LIN {X 0,Y 531.686,Z 941.292,A -85,B 0,C 180,E1 4384.403,E2 4384.403} C_VEL
LIN {X 0,Y 531.304,Z 953.867,A -85,B 0,C 180,E1 4387.483,E2 4387.483} C_VEL
LIN {X 0,Y 531.16,Z 959.735,A -85,B 0,C 180,E1 4390.034,E2 4390.034} C_VEL
LIN {X 0,Y 530.961,Z 961.944,A -85,B 0,C 180,E1 4393.431,E2 4393.431} C_VEL
LIN {X 0,Y 531.167,Z 959.168,A -85,B 0,C 180,E1 4396.197,E2 4396.197} C_VEL
LIN {X 0,Y 531.42,Z 951.627,A -85,B 0,C 180,E1 4399.095,E2 4399.095} C_VEL
LIN {X 0,Y 531.761,Z 938.386,A -85,B 0,C 180,E1 4402.021,E2 4402.021} C_VEL
LIN {X 0,Y 532.428,Z 919.705,A -85,B 0,C 180,E1 4404.691,E2 4404.691} C_VEL
LIN {X 0,Y 533.219,Z 897.252,A -85,B 0,C 180,E1 4406.846,E2 4406.846} C_VEL
LIN {X 0,Y 533.797,Z 871.722,A -85,B 0,C 180,E1 4408.476,E2 4408.476} C_VEL
LIN {X 0,Y 530.532,Z 857.28,A -85,B 0,C 180,E1 4409.284,E2 4409.284} C_VEL
LIN {X 0,Y 530.829,Z 857.28,A -85,B 0,C 180,E1 4414.908,E2 4414.908} C_VEL
LIN {X 0,Y 530.721,Z 857.28,A -85,B 0,C 180,E1 4419.855,E2 4419.855} C_VEL
LIN {X 0,Y 530.626,Z 857.28,A -85,B 0,C 180,E1 4424.88,E2 4424.88} C_VEL
LIN {X 0,Y 530.545,Z 857.28,A -85,B 0,C 180,E1 4430.026,E2 4430.026} C_VEL
LIN {X 0,Y 530.38,Z 857.28,A -85,B 0,C 180,E1 4435.353,E2 4435.353} C_VEL
LIN {X 0,Y 530.253,Z 857.28,A -85,B 0,C 180,E1 4441.143,E2 4441.143} C_VEL
LIN {X 0,Y 530.208,Z 857.28,A -85,B 0,C 180,E1 4446.978,E2 4446.978} C_VEL
LIN {X 0,Y 530.229,Z 857.28,A -85,B 0,C 180,E1 4453.26,E2 4453.26} C_VEL
LIN {X 0,Y 530.267,Z 857.28,A -85,B 0,C 180,E1 4458.999,E2 4458.999} C_VEL
LIN {X 0,Y 530.449,Z 857.934,A -85,B 0,C 180,E1 4461.861,E2 4461.861} C_VEL
LIN {X 0,Y 533.507,Z 877.785,A -85,B 0,C 180,E1 4462.888,E2 4462.888} C_VEL
LIN {X 0,Y 532.84,Z 903.715,A -85,B 0,C 180,E1 4464.706,E2 4464.706} C_VEL
LIN {X 0,Y 532.072,Z 925.667,A -85,B 0,C 180,E1 4467.04,E2 4467.04} C_VEL
LIN {X 0,Y 531.58,Z 942.941,A -85,B 0,C 180,E1 4469.823,E2 4469.823} C_VEL
LIN {X 0,Y 531.314,Z 954.833,A -85,B 0,C 180,E1 4472.91,E2 4472.91} C_VEL
LIN {X 0,Y 531.021,Z 960.608,A -85,B 0,C 180,E1 4475.838,E2 4475.838} C_VEL
LIN {X 0,Y 530.948,Z 961.777,A -85,B 0,C 180,E1 4478.273,E2 4478.273} C_VEL
LIN {X 0,Y 531.171,Z 959.373,A -85,B 0,C 180,E1 4480.97,E2 4480.97} C_VEL
LIN {X 0,Y 531.35,Z 952.112,A -85,B 0,C 180,E1 4483.898,E2 4483.898} C_VEL
LIN {X 0,Y 531.721,Z 939.03,A -85,B 0,C 180,E1 4486.86,E2 4486.86} C_VEL
LIN {X 0,Y 532.237,Z 921.058,A -85,B 0,C 180,E1 4489.473,E2 4489.473} C_VEL
LIN {X 0,Y 532.958,Z 898.658,A -85,B 0,C 180,E1 4491.653,E2 4491.653} C_VEL
LIN {X 0,Y 533.718,Z 872.183,A -85,B 0,C 180,E1 4493.332,E2 4493.332} C_VEL
LIN {X 0,Y 530.984,Z 857.28,A -85,B 0,C 180,E1 4494.148,E2 4494.148} C_VEL
LIN {X 0,Y 530.827,Z 857.28,A -85,B 0,C 180,E1 4500.021,E2 4500.021} C_VEL
LIN {X 0,Y 530.801,Z 857.28,A -85,B 0,C 180,E1 4504.928,E2 4504.928} C_VEL
LIN {X 0,Y 530.696,Z 857.28,A -85,B 0,C 180,E1 4509.873,E2 4509.873} C_VEL
LIN {X 0,Y 530.612,Z 857.28,A -85,B 0,C 180,E1 4514.896,E2 4514.896} C_VEL
LIN {X 0,Y 530.576,Z 857.28,A -85,B 0,C 180,E1 4520.039,E2 4520.039} C_VEL
LIN {X 0,Y 530.461,Z 857.28,A -85,B 0,C 180,E1 4525.361,E2 4525.361} C_VEL
LIN {X 0,Y 530.352,Z 857.28,A -85,B 0,C 180,E1 4527.012,E2 4527.012} C_VEL
LIN {X 0,Y 527.829,Z 857.28,A -85,B 0,C 180,E1 4528.404,E2 4528.404} C_VEL
LIN {X 0,Y 522.406,Z 857.28,A -85,B 0,C 180,E1 4530.49,E2 4530.49} C_VEL
LIN {X 0,Y 522.316,Z 857.28,A -85,B 0,C 180,E1 4530.731,E2 4530.731} C_VEL
LIN {X 0,Y 522.326,Z 857.28,A -85,B 0,C 180,E1 4535.744,E2 4535.744} C_VEL
LIN {X 0,Y 522.316,Z 857.28,A -85,B 0,C 180,E1 4541.821,E2 4541.821} C_VEL
LIN {X 0,Y 522.421,Z 857.28,A -85,B 0,C 180,E1 4548.197,E2 4548.197} C_VEL
LIN {X 0,Y 522.325,Z 857.28,A -85,B 0,C 180,E1 4554.568,E2 4554.568} C_VEL
LIN {X 0,Y 522.426,Z 857.28,A -85,B 0,C 180,E1 4560.483,E2 4560.483} C_VEL
LIN {X 0,Y 522.61,Z 857.28,A -85,B 0,C 180,E1 4564.312,E2 4564.312} C_VEL
LIN {X 0,Y 530.423,Z 879.508,A -85,B 0,C 180,E1 4565.071,E2 4565.071} C_VEL
LIN {X 0,Y 530.037,Z 939.927,A -85,B 0,C 180,E1 4566.073,E2 4566.073} C_VEL
LIN {X 0,Y 528.959,Z 972.429,A -85,B 0,C 180,E1 4567.213,E2 4567.213} C_VEL
LIN {X 0,Y 527.599,Z 1004.287,A -85,B 0,C 180,E1 4568.993,E2 4568.993} C_VEL
LIN {X 0,Y 526.123,Z 1033.257,A -85,B 0,C 180,E1 4571.328,E2 4571.328} C_VEL
LIN {X 0,Y 524.904,Z 1058.08,A -85,B 0,C 180,E1 4574.097,E2 4574.097} C_VEL
LIN {X 0,Y 523.978,Z 1078.839,A -85,B 0,C 180,E1 4577.272,E2 4577.272} C_VEL
LIN {X 0,Y 523.47,Z 1095.118,A -85,B 0,C 180,E1 4580.847,E2 4580.847} C_VEL
LIN {X 0,Y 523.252,Z 1104.993,A -85,B 0,C 180,E1 4584.188,E2 4584.188} C_VEL
LIN {X 0,Y 523.184,Z 1109.404,A -85,B 0,C 180,E1 4586.682,E2 4586.682} C_VEL
LIN {X 0,Y 523.198,Z 1111.5,A -85,B 0,C 180,E1 4590.001,E2 4590.001} C_VEL
LIN {X 0,Y 523.22,Z 1108.484,A -85,B 0,C 180,E1 4593.955,E2 4593.955} C_VEL
LIN {X 0,Y 523.378,Z 1100.701,A -85,B 0,C 180,E1 4597.481,E2 4597.481} C_VEL
LIN {X 0,Y 523.696,Z 1087.408,A -85,B 0,C 180,E1 4601.022,E2 4601.022} C_VEL
LIN {X 0,Y 524.459,Z 1068.424,A -85,B 0,C 180,E1 4604.456,E2 4604.456} C_VEL
LIN {X 0,Y 525.575,Z 1043.869,A -85,B 0,C 180,E1 4607.594,E2 4607.594} C_VEL
LIN {X 0,Y 526.962,Z 1015.854,A -85,B 0,C 180,E1 4610.169,E2 4610.169} C_VEL
LIN {X 0,Y 528.484,Z 984.528,A -85,B 0,C 180,E1 4612.199,E2 4612.199} C_VEL
LIN {X 0,Y 529.692,Z 950.575,A -85,B 0,C 180,E1 4613.623,E2 4613.623} C_VEL
LIN {X 0,Y 530.348,Z 915.537,A -85,B 0,C 180,E1 4614.406,E2 4614.406} C_VEL
LIN {X 0,Y 529.868,Z 878.299,A -85,B 0,C 180,E1 4614.974,E2 4614.974} C_VEL
LIN {X 0,Y 522.471,Z 857.28,A -85,B 0,C 180,E1 4615.766,E2 4615.766} C_VEL
LIN {X 0,Y 522.371,Z 857.28,A -85,B 0,C 180,E1 4621.449,E2 4621.449} C_VEL
LIN {X 0,Y 522.284,Z 857.28,A -85,B 0,C 180,E1 4627.502,E2 4627.502} C_VEL
LIN {X 0,Y 522.319,Z 857.28,A -85,B 0,C 180,E1 4633.552,E2 4633.552} C_VEL
LIN {X 0,Y 522.389,Z 857.28,A -85,B 0,C 180,E1 4638.902,E2 4638.902} C_VEL
LIN {X 0,Y 522.342,Z 857.28,A -85,B 0,C 180,E1 4644.56,E2 4644.56} C_VEL
LIN {X 0,Y 522.409,Z 857.28,A -85,B 0,C 180,E1 4650.471,E2 4650.471} C_VEL
LIN {X 0,Y 522.582,Z 857.28,A -85,B 0,C 180,E1 4656.058,E2 4656.058} C_VEL
LIN {X 0,Y 522.722,Z 857.28,A -85,B 0,C 180,E1 4661.407,E2 4661.407} C_VEL
LIN {X 0,Y 522.636,Z 857.28,A -85,B 0,C 180,E1 4668.283,E2 4668.283} C_VEL
LIN {X 0,Y 522.958,Z 857.28,A -85,B 0,C 180,E1 4673.331,E2 4673.331} C_VEL
LIN {X 0,Y 522.942,Z 857.28,A -85,B 0,C 180,E1 4679.979,E2 4679.979} C_VEL
LIN {X 0,Y 522.877,Z 857.28,A -85,B 0,C 180,E1 4684.96,E2 4684.96} C_VEL
LIN {X 0,Y 522.769,Z 857.28,A -85,B 0,C 180,E1 4690.022,E2 4690.022} C_VEL
LIN {X 0,Y 522.692,Z 857.28,A -85,B 0,C 180,E1 4695.083,E2 4695.083} C_VEL
LIN {X 0,Y 522.637,Z 857.28,A -85,B 0,C 180,E1 4700.311,E2 4700.311} C_VEL
LIN {X 0,Y 522.478,Z 857.28,A -85,B 0,C 180,E1 4706.058,E2 4706.058} C_VEL
LIN {X 0,Y 522.342,Z 857.28,A -85,B 0,C 180,E1 4711.41,E2 4711.41} C_VEL
LIN {X 0,Y 522.255,Z 857.28,A -85,B 0,C 180,E1 4717.458,E2 4717.458} C_VEL
LIN {X 0,Y 522.35,Z 857.28,A -85,B 0,C 180,E1 4723.56,E2 4723.56} C_VEL
LIN {X 0,Y 522.376,Z 857.28,A -85,B 0,C 180,E1 4728.842,E2 4728.842} C_VEL
LIN {X 0,Y 522.429,Z 857.28,A -85,B 0,C 180,E1 4734.575,E2 4734.575} C_VEL
LIN {X 0,Y 522.636,Z 857.79,A -85,B 0,C 180,E1 4736.295,E2 4736.295} C_VEL
LIN {X 0,Y 526.502,Z 877.686,A -85,B 0,C 180,E1 4737.414,E2 4737.414} C_VEL
LIN {X 0,Y 525.643,Z 903.07,A -85,B 0,C 180,E1 4739.199,E2 4739.199} C_VEL
LIN {X 0,Y 524.669,Z 924.663,A -85,B 0,C 180,E1 4741.464,E2 4741.464} C_VEL
LIN {X 0,Y 524.04,Z 941.697,A -85,B 0,C 180,E1 4744.104,E2 4744.104} C_VEL
LIN {X 0,Y 523.64,Z 953.648,A -85,B 0,C 180,E1 4746.937,E2 4746.937} C_VEL
LIN {X 0,Y 523.4,Z 960.427,A -85,B 0,C 180,E1 4749.687,E2 4749.687} C_VEL
LIN {X 0,Y 523.152,Z 963.153,A -85,B 0,C 180,E1 4752.608,E2 4752.608} C_VEL
LIN {X 0,Y 523.311,Z 961.505,A -85,B 0,C 180,E1 4755.481,E2 4755.481} C_VEL
LIN {X 0,Y 523.516,Z 955.588,A -85,B 0,C 180,E1 4758.319,E2 4758.319} C_VEL
LIN {X 0,Y 523.978,Z 943.155,A -85,B 0,C 180,E1 4761.483,E2 4761.483} C_VEL
LIN {X 0,Y 524.612,Z 925.67,A -85,B 0,C 180,E1 4764.282,E2 4764.282} C_VEL
LIN {X 0,Y 525.495,Z 904.106,A -85,B 0,C 180,E1 4766.593,E2 4766.593} C_VEL
LIN {X 0,Y 526.42,Z 879.629,A -85,B 0,C 180,E1 4768.351,E2 4768.351} C_VEL
LIN {X 0,Y 524.585,Z 865.354,A -85,B 0,C 180,E1 4769.173,E2 4769.173} C_VEL
LIN {X 0,Y 522.578,Z 857.28,A -85,B 0,C 180,E1 4769.688,E2 4769.688} C_VEL
LIN {X 0,Y 522.915,Z 857.28,A -85,B 0,C 180,E1 4774.983,E2 4774.983} C_VEL
LIN {X 0,Y 522.774,Z 857.28,A -85,B 0,C 180,E1 4780.288,E2 4780.288} C_VEL
LIN {X 0,Y 522.689,Z 857.28,A -85,B 0,C 180,E1 4785.111,E2 4785.111} C_VEL
LIN {X 0,Y 522.592,Z 857.28,A -85,B 0,C 180,E1 4790.344,E2 4790.344} C_VEL
LIN {X 0,Y 522.426,Z 857.28,A -85,B 0,C 180,E1 4796.146,E2 4796.146} C_VEL
LIN {X 0,Y 522.344,Z 857.28,A -85,B 0,C 180,E1 4801.449,E2 4801.449} C_VEL
LIN {X 0,Y 522.245,Z 857.28,A -85,B 0,C 180,E1 4807.504,E2 4807.504} C_VEL
LIN {X 0,Y 522.328,Z 857.28,A -85,B 0,C 180,E1 4813.615,E2 4813.615} C_VEL
LIN {X 0,Y 522.374,Z 857.28,A -85,B 0,C 180,E1 4818.902,E2 4818.902} C_VEL
LIN {X 0,Y 522.476,Z 857.505,A -85,B 0,C 180,E1 4821.573,E2 4821.573} C_VEL
LIN {X 0,Y 525.93,Z 878.07,A -85,B 0,C 180,E1 4822.641,E2 4822.641} C_VEL
LIN {X 0,Y 525.266,Z 903.689,A -85,B 0,C 180,E1 4824.434,E2 4824.434} C_VEL
LIN {X 0,Y 524.418,Z 925.824,A -85,B 0,C 180,E1 4826.773,E2 4826.773} C_VEL
LIN {X 0,Y 523.86,Z 942.873,A -85,B 0,C 180,E1 4829.473,E2 4829.473} C_VEL
LIN {X 0,Y 523.539,Z 954.889,A -85,B 0,C 180,E1 4832.474,E2 4832.474} C_VEL
LIN {X 0,Y 523.261,Z 961.323,A -85,B 0,C 180,E1 4835.456,E2 4835.456} C_VEL
LIN {X 0,Y 523.151,Z 963.019,A -85,B 0,C 180,E1 4837.932,E2 4837.932} C_VEL
LIN {X 0,Y 523.343,Z 961.014,A -85,B 0,C 180,E1 4840.722,E2 4840.722} C_VEL
LIN {X 0,Y 523.558,Z 954.393,A -85,B 0,C 180,E1 4843.652,E2 4843.652} C_VEL
LIN {X 0,Y 523.892,Z 942.002,A -85,B 0,C 180,E1 4846.66,E2 4846.66} C_VEL
LIN {X 0,Y 524.514,Z 924.374,A -85,B 0,C 180,E1 4849.37,E2 4849.37} C_VEL
LIN {X 0,Y 525.279,Z 902.377,A -85,B 0,C 180,E1 4851.634,E2 4851.634} C_VEL
LIN {X 0,Y 526.144,Z 877.428,A -85,B 0,C 180,E1 4853.325,E2 4853.325} C_VEL
LIN {X 0,Y 523.03,Z 857.28,A -85,B 0,C 180,E1 4854.417,E2 4854.417} C_VEL
LIN {X 0,Y 522.945,Z 857.28,A -85,B 0,C 180,E1 4860.021,E2 4860.021} C_VEL
LIN {X 0,Y 522.887,Z 857.28,A -85,B 0,C 180,E1 4865.003,E2 4865.003} C_VEL
LIN {X 0,Y 522.792,Z 857.28,A -85,B 0,C 180,E1 4870.043,E2 4870.043} C_VEL
LIN {X 0,Y 522.676,Z 857.28,A -85,B 0,C 180,E1 4875.127,E2 4875.127} C_VEL
LIN {X 0,Y 522.636,Z 857.28,A -85,B 0,C 180,E1 4880.356,E2 4880.356} C_VEL
LIN {X 0,Y 522.462,Z 857.28,A -85,B 0,C 180,E1 4886.057,E2 4886.057} C_VEL
LIN {X 0,Y 522.316,Z 857.28,A -85,B 0,C 180,E1 4890.731,E2 4890.731} C_VEL
LIN {X 0,Y 519.814,Z 857.28,A -85,B 0,C 180,E1 4892.139,E2 4892.139} C_VEL
LIN {X 0,Y 514.508,Z 857.28,A -85,B 0,C 180,E1 4894.249,E2 4894.249} C_VEL
LIN {X 0,Y 514.42,Z 857.28,A -85,B 0,C 180,E1 4894.493,E2 4894.493} C_VEL
LIN {X 0,Y 514.38,Z 857.28,A -85,B 0,C 180,E1 4900.366,E2 4900.366} C_VEL
LIN {X 0,Y 514.435,Z 857.28,A -85,B 0,C 180,E1 4905.061,E2 4905.061} C_VEL
LIN {X 0,Y 514.493,Z 857.28,A -85,B 0,C 180,E1 4909.924,E2 4909.924} C_VEL
LIN {X 0,Y 514.394,Z 857.28,A -85,B 0,C 180,E1 4915.997,E2 4915.997} C_VEL
LIN {X 0,Y 514.572,Z 857.28,A -85,B 0,C 180,E1 4921.972,E2 4921.972} C_VEL
LIN {X 0,Y 514.678,Z 857.28,A -85,B 0,C 180,E1 4923.935,E2 4923.935} C_VEL
LIN {X 0,Y 523.207,Z 881.258,A -85,B 0,C 180,E1 4924.73,E2 4924.73} C_VEL
LIN {X 0,Y 522.815,Z 939.926,A -85,B 0,C 180,E1 4925.722,E2 4925.722} C_VEL
LIN {X 0,Y 521.638,Z 972.428,A -85,B 0,C 180,E1 4926.875,E2 4926.875} C_VEL
LIN {X 0,Y 520.147,Z 1004.749,A -85,B 0,C 180,E1 4928.711,E2 4928.711} C_VEL
LIN {X 0,Y 518.481,Z 1034.401,A -85,B 0,C 180,E1 4931.153,E2 4931.153} C_VEL
LIN {X 0,Y 517.127,Z 1059.679,A -85,B 0,C 180,E1 4934.069,E2 4934.069} C_VEL
LIN {X 0,Y 516.104,Z 1081.097,A -85,B 0,C 180,E1 4937.505,E2 4937.505} C_VEL
LIN {X 0,Y 515.593,Z 1096.65,A -85,B 0,C 180,E1 4941.132,E2 4941.132} C_VEL
LIN {X 0,Y 515.398,Z 1106.726,A -85,B 0,C 180,E1 4944.945,E2 4944.945} C_VEL
LIN {X 0,Y 515.284,Z 1110.932,A -85,B 0,C 180,E1 4948.317,E2 4948.317} C_VEL
LIN {X 0,Y 515.293,Z 1110.931,A -85,B 0,C 180,E1 4951.684,E2 4951.684} C_VEL
LIN {X 0,Y 515.399,Z 1106.723,A -85,B 0,C 180,E1 4955.057,E2 4955.057} C_VEL
LIN {X 0,Y 515.605,Z 1096.648,A -85,B 0,C 180,E1 4958.869,E2 4958.869} C_VEL
LIN {X 0,Y 516.101,Z 1081.092,A -85,B 0,C 180,E1 4962.496,E2 4962.496} C_VEL
LIN {X 0,Y 517.137,Z 1059.67,A -85,B 0,C 180,E1 4965.932,E2 4965.932} C_VEL
LIN {X 0,Y 518.503,Z 1034.387,A -85,B 0,C 180,E1 4968.847,E2 4968.847} C_VEL
LIN {X 0,Y 520.158,Z 1004.698,A -85,B 0,C 180,E1 4971.292,E2 4971.292} C_VEL
LIN {X 0,Y 521.592,Z 972.395,A -85,B 0,C 180,E1 4973.129,E2 4973.129} C_VEL
LIN {X 0,Y 522.793,Z 937.798,A -85,B 0,C 180,E1 4974.341,E2 4974.341} C_VEL
LIN {X 0,Y 522.824,Z 880.394,A -85,B 0,C 180,E1 4975.303,E2 4975.303} C_VEL
LIN {X 0,Y 514.56,Z 857.28,A -85,B 0,C 180,E1 4976.12,E2 4976.12} C_VEL
LIN {X 0,Y 514.453,Z 857.28,A -85,B 0,C 180,E1 4981.99,E2 4981.99} C_VEL
LIN {X 0,Y 514.363,Z 857.28,A -85,B 0,C 180,E1 4988.182,E2 4988.182} C_VEL
LIN {X 0,Y 514.366,Z 857.28,A -85,B 0,C 180,E1 4992.612,E2 4992.612} C_VEL
LIN {X 0,Y 514.446,Z 857.28,A -85,B 0,C 180,E1 4997.39,E2 4997.39} C_VEL
LIN {X 0,Y 514.434,Z 857.28,A -85,B 0,C 180,E1 5002.624,E2 5002.624} C_VEL
LIN {X 0,Y 514.48,Z 857.28,A -85,B 0,C 180,E1 5008.59,E2 5008.59} C_VEL
LIN {X 0,Y 514.578,Z 857.28,A -85,B 0,C 180,E1 5013.798,E2 5013.798} C_VEL
LIN {X 0,Y 514.739,Z 857.28,A -85,B 0,C 180,E1 5020.267,E2 5020.267} C_VEL
LIN {X 0,Y 514.565,Z 857.28,A -85,B 0,C 180,E1 5026.172,E2 5026.172} C_VEL
LIN {X 0,Y 514.82,Z 857.28,A -85,B 0,C 180,E1 5031.526,E2 5031.526} C_VEL
LIN {X 0,Y 514.981,Z 857.28,A -85,B 0,C 180,E1 5036.609,E2 5036.609} C_VEL
LIN {X 0,Y 514.972,Z 857.28,A -85,B 0,C 180,E1 5041.663,E2 5041.663} C_VEL
LIN {X 0,Y 514.904,Z 857.28,A -85,B 0,C 180,E1 5046.73,E2 5046.73} C_VEL
LIN {X 0,Y 514.781,Z 857.28,A -85,B 0,C 180,E1 5051.854,E2 5051.854} C_VEL
LIN {X 0,Y 514.737,Z 857.28,A -85,B 0,C 180,E1 5057.076,E2 5057.076} C_VEL
LIN {X 0,Y 514.634,Z 857.28,A -85,B 0,C 180,E1 5062.453,E2 5062.453} C_VEL
LIN {X 0,Y 514.526,Z 857.28,A -85,B 0,C 180,E1 5068.05,E2 5068.05} C_VEL
LIN {X 0,Y 514.385,Z 857.28,A -85,B 0,C 180,E1 5073.962,E2 5073.962} C_VEL
LIN {X 0,Y 514.382,Z 857.28,A -85,B 0,C 180,E1 5080.309,E2 5080.309} C_VEL
LIN {X 0,Y 514.406,Z 857.28,A -85,B 0,C 180,E1 5085.056,E2 5085.056} C_VEL
LIN {X 0,Y 514.464,Z 857.28,A -85,B 0,C 180,E1 5091.827,E2 5091.827} C_VEL
LIN {X 0,Y 514.722,Z 857.28,A -85,B 0,C 180,E1 5095.905,E2 5095.905} C_VEL
LIN {X 0,Y 519.052,Z 878.103,A -85,B 0,C 180,E1 5097.103,E2 5097.103} C_VEL
LIN {X 0,Y 518.142,Z 903.526,A -85,B 0,C 180,E1 5098.901,E2 5098.901} C_VEL
LIN {X 0,Y 517.103,Z 925.104,A -85,B 0,C 180,E1 5101.175,E2 5101.175} C_VEL
LIN {X 0,Y 516.343,Z 942.645,A -85,B 0,C 180,E1 5103.905,E2 5103.905} C_VEL
LIN {X 0,Y 515.932,Z 954.252,A -85,B 0,C 180,E1 5106.66,E2 5106.66} C_VEL
LIN {X 0,Y 515.589,Z 962.018,A -85,B 0,C 180,E1 5109.872,E2 5109.872} C_VEL
LIN {X 0,Y 515.372,Z 964.38,A -85,B 0,C 180,E1 5112.915,E2 5112.915} C_VEL
LIN {X 0,Y 515.584,Z 961.302,A -85,B 0,C 180,E1 5116.412,E2 5116.412} C_VEL
LIN {X 0,Y 515.929,Z 953.427,A -85,B 0,C 180,E1 5119.443,E2 5119.443} C_VEL
LIN {X 0,Y 516.389,Z 940.148,A -85,B 0,C 180,E1 5122.418,E2 5122.418} C_VEL
LIN {X 0,Y 517.248,Z 921.213,A -85,B 0,C 180,E1 5125.172,E2 5125.172} C_VEL
LIN {X 0,Y 518.229,Z 898.544,A -85,B 0,C 180,E1 5127.383,E2 5127.383} C_VEL
LIN {X 0,Y 518.522,Z 873.107,A -85,B 0,C 180,E1 5129.058,E2 5129.058} C_VEL
LIN {X 0,Y 514.633,Z 857.28,A -85,B 0,C 180,E1 5129.999,E2 5129.999} C_VEL
LIN {X 0,Y 515.018,Z 857.28,A -85,B 0,C 180,E1 5135.059,E2 5135.059} C_VEL
LIN {X 0,Y 514.896,Z 857.28,A -85,B 0,C 180,E1 5140.161,E2 5140.161} C_VEL
LIN {X 0,Y 514.751,Z 857.28,A -85,B 0,C 180,E1 5145.35,E2 5145.35} C_VEL
LIN {X 0,Y 514.648,Z 857.28,A -85,B 0,C 180,E1 5150.673,E2 5150.673} C_VEL
LIN {X 0,Y 514.546,Z 857.28,A -85,B 0,C 180,E1 5156.191,E2 5156.191} C_VEL
LIN {X 0,Y 514.428,Z 857.28,A -85,B 0,C 180,E1 5161.99,E2 5161.99} C_VEL
LIN {X 0,Y 514.344,Z 857.28,A -85,B 0,C 180,E1 5168.183,E2 5168.183} C_VEL
LIN {X 0,Y 514.394,Z 857.28,A -85,B 0,C 180,E1 5174.944,E2 5174.944} C_VEL
LIN {X 0,Y 514.622,Z 858.024,A -85,B 0,C 180,E1 5181.318,E2 5181.318} C_VEL
LIN {X 0,Y 518.349,Z 879.334,A -85,B 0,C 180,E1 5182.443,E2 5182.443} C_VEL
LIN {X 0,Y 517.635,Z 904.658,A -85,B 0,C 180,E1 5184.242,E2 5184.242} C_VEL
LIN {X 0,Y 516.804,Z 925.31,A -85,B 0,C 180,E1 5186.416,E2 5186.416} C_VEL
LIN {X 0,Y 516.172,Z 941.896,A -85,B 0,C 180,E1 5188.955,E2 5188.955} C_VEL
LIN {X 0,Y 515.766,Z 954.888,A -85,B 0,C 180,E1 5192.023,E2 5192.023} C_VEL
LIN {X 0,Y 515.548,Z 961.578,A -85,B 0,C 180,E1 5194.804,E2 5194.804} C_VEL
LIN {X 0,Y 515.323,Z 964.146,A -85,B 0,C 180,E1 5197.579,E2 5197.579} C_VEL
LIN {X 0,Y 515.481,Z 963.124,A -85,B 0,C 180,E1 5200.034,E2 5200.034} C_VEL
LIN {X 0,Y 515.741,Z 957.805,A -85,B 0,C 180,E1 5202.958,E2 5202.958} C_VEL
LIN {X 0,Y 516.086,Z 947.027,A -85,B 0,C 180,E1 5206,E2 5206} C_VEL
LIN {X 0,Y 516.68,Z 930.919,A -85,B 0,C 180,E1 5208.812,E2 5208.812} C_VEL
LIN {X 0,Y 517.521,Z 909.442,A -85,B 0,C 180,E1 5211.296,E2 5211.296} C_VEL
LIN {X 0,Y 518.354,Z 885.382,A -85,B 0,C 180,E1 5213.144,E2 5213.144} C_VEL
LIN {X 0,Y 517.545,Z 868.672,A -85,B 0,C 180,E1 5214.076,E2 5214.076} C_VEL
LIN {X 0,Y 515.108,Z 857.28,A -85,B 0,C 180,E1 5214.656,E2 5214.656} C_VEL
LIN {X 0,Y 515.044,Z 857.28,A -85,B 0,C 180,E1 5220.022,E2 5220.022} C_VEL
LIN {X 0,Y 514.98,Z 857.28,A -85,B 0,C 180,E1 5225.08,E2 5225.08} C_VEL
LIN {X 0,Y 514.896,Z 857.28,A -85,B 0,C 180,E1 5230.179,E2 5230.179} C_VEL
LIN {X 0,Y 514.767,Z 857.28,A -85,B 0,C 180,E1 5235.366,E2 5235.366} C_VEL
LIN {X 0,Y 514.701,Z 857.28,A -85,B 0,C 180,E1 5240.685,E2 5240.685} C_VEL
LIN {X 0,Y 514.557,Z 857.28,A -85,B 0,C 180,E1 5246.203,E2 5246.203} C_VEL
LIN {X 0,Y 514.462,Z 857.28,A -85,B 0,C 180,E1 5251.998,E2 5251.998} C_VEL
LIN {X 0,Y 514.42,Z 857.28,A -85,B 0,C 180,E1 5254.493,E2 5254.493} C_VEL
LIN {X 0,Y 511.854,Z 857.28,A -85,B 0,C 180,E1 5255.93,E2 5255.93} C_VEL
LIN {X 0,Y 506.441,Z 857.28,A -85,B 0,C 180,E1 5258.083,E2 5258.083} C_VEL
LIN {X 0,Y 506.357,Z 857.28,A -85,B 0,C 180,E1 5258.333,E2 5258.333} C_VEL
LIN {X 0,Y 506.432,Z 857.28,A -85,B 0,C 180,E1 5264.15,E2 5264.15} C_VEL
LIN {X 0,Y 506.496,Z 857.28,A -85,B 0,C 180,E1 5268.88,E2 5268.88} C_VEL
LIN {X 0,Y 506.484,Z 857.28,A -85,B 0,C 180,E1 5275.391,E2 5275.391} C_VEL
LIN {X 0,Y 506.589,Z 857.28,A -85,B 0,C 180,E1 5281.433,E2 5281.433} C_VEL
LIN {X 0,Y 506.719,Z 857.28,A -85,B 0,C 180,E1 5283.563,E2 5283.563} C_VEL
LIN {X 0,Y 516.179,Z 885.355,A -85,B 0,C 180,E1 5284.423,E2 5284.423} C_VEL
LIN {X 0,Y 515.581,Z 941.148,A -85,B 0,C 180,E1 5285.394,E2 5285.394} C_VEL
LIN {X 0,Y 514.28,Z 974.856,A -85,B 0,C 180,E1 5286.639,E2 5286.639} C_VEL
LIN {X 0,Y 512.594,Z 1006.805,A -85,B 0,C 180,E1 5288.534,E2 5288.534} C_VEL
LIN {X 0,Y 510.831,Z 1035.498,A -85,B 0,C 180,E1 5290.972,E2 5290.972} C_VEL
LIN {X 0,Y 509.354,Z 1061.277,A -85,B 0,C 180,E1 5294.041,E2 5294.041} C_VEL
LIN {X 0,Y 508.243,Z 1082.183,A -85,B 0,C 180,E1 5297.528,E2 5297.528} C_VEL
LIN {X 0,Y 507.722,Z 1096.65,A -85,B 0,C 180,E1 5300.993,E2 5300.993} C_VEL
LIN {X 0,Y 507.492,Z 1106.725,A -85,B 0,C 180,E1 5304.866,E2 5304.866} C_VEL
LIN {X 0,Y 507.401,Z 1110.932,A -85,B 0,C 180,E1 5308.291,E2 5308.291} C_VEL
LIN {X 0,Y 507.409,Z 1110.931,A -85,B 0,C 180,E1 5311.711,E2 5311.711} C_VEL
LIN {X 0,Y 507.493,Z 1106.723,A -85,B 0,C 180,E1 5315.136,E2 5315.136} C_VEL
LIN {X 0,Y 507.735,Z 1096.648,A -85,B 0,C 180,E1 5319.008,E2 5319.008} C_VEL
LIN {X 0,Y 508.286,Z 1081.092,A -85,B 0,C 180,E1 5322.691,E2 5322.691} C_VEL
LIN {X 0,Y 509.414,Z 1059.67,A -85,B 0,C 180,E1 5326.18,E2 5326.18} C_VEL
LIN {X 0,Y 510.931,Z 1034.388,A -85,B 0,C 180,E1 5329.137,E2 5329.137} C_VEL
LIN {X 0,Y 512.698,Z 1005.302,A -85,B 0,C 180,E1 5331.573,E2 5331.573} C_VEL
LIN {X 0,Y 514.308,Z 972.393,A -85,B 0,C 180,E1 5333.476,E2 5333.476} C_VEL
LIN {X 0,Y 515.627,Z 937.222,A -85,B 0,C 180,E1 5334.717,E2 5334.717} C_VEL
LIN {X 0,Y 515.82,Z 882.841,A -85,B 0,C 180,E1 5335.633,E2 5335.633} C_VEL
LIN {X 0,Y 506.612,Z 857.28,A -85,B 0,C 180,E1 5336.511,E2 5336.511} C_VEL
LIN {X 0,Y 506.479,Z 857.28,A -85,B 0,C 180,E1 5342.555,E2 5342.555} C_VEL
LIN {X 0,Y 506.479,Z 857.28,A -85,B 0,C 180,E1 5346.719,E2 5346.719} C_VEL
LIN {X 0,Y 506.375,Z 857.28,A -85,B 0,C 180,E1 5353.45,E2 5353.45} C_VEL
LIN {X 0,Y 506.471,Z 857.28,A -85,B 0,C 180,E1 5358.869,E2 5358.869} C_VEL
LIN {X 0,Y 506.5,Z 857.28,A -85,B 0,C 180,E1 5365.382,E2 5365.382} C_VEL
LIN {X 0,Y 506.53,Z 857.28,A -85,B 0,C 180,E1 5371.417,E2 5371.417} C_VEL
LIN {X 0,Y 506.746,Z 857.28,A -85,B 0,C 180,E1 5377.131,E2 5377.131} C_VEL
LIN {X 0,Y 506.876,Z 857.28,A -85,B 0,C 180,E1 5382.916,E2 5382.916} C_VEL
LIN {X 0,Y 506.899,Z 857.28,A -85,B 0,C 180,E1 5389.658,E2 5389.658} C_VEL
LIN {X 0,Y 507.094,Z 857.28,A -85,B 0,C 180,E1 5394.841,E2 5394.841} C_VEL
LIN {X 0,Y 507.191,Z 857.28,A -85,B 0,C 180,E1 5399.978,E2 5399.978} C_VEL
LIN {X 0,Y 507.056,Z 857.28,A -85,B 0,C 180,E1 5405.115,E2 5405.115} C_VEL
LIN {X 0,Y 506.972,Z 857.28,A -85,B 0,C 180,E1 5410.296,E2 5410.296} C_VEL
LIN {X 0,Y 506.841,Z 857.28,A -85,B 0,C 180,E1 5415.566,E2 5415.566} C_VEL
LIN {X 0,Y 506.767,Z 857.28,A -85,B 0,C 180,E1 5420.977,E2 5420.977} C_VEL
LIN {X 0,Y 506.638,Z 857.28,A -85,B 0,C 180,E1 5426.596,E2 5426.596} C_VEL
LIN {X 0,Y 506.468,Z 857.28,A -85,B 0,C 180,E1 5432.513,E2 5432.513} C_VEL
LIN {X 0,Y 506.411,Z 857.28,A -85,B 0,C 180,E1 5438.844,E2 5438.844} C_VEL
LIN {X 0,Y 506.406,Z 857.28,A -85,B 0,C 180,E1 5444.145,E2 5444.145} C_VEL
LIN {X 0,Y 506.452,Z 857.28,A -85,B 0,C 180,E1 5448.874,E2 5448.874} C_VEL
LIN {X 0,Y 506.762,Z 857.552,A -85,B 0,C 180,E1 5455.547,E2 5455.547} C_VEL
LIN {X 0,Y 511.666,Z 879.946,A -85,B 0,C 180,E1 5456.87,E2 5456.87} C_VEL
LIN {X 0,Y 510.646,Z 905.344,A -85,B 0,C 180,E1 5458.716,E2 5458.716} C_VEL
LIN {X 0,Y 509.48,Z 927.135,A -85,B 0,C 180,E1 5461.079,E2 5461.079} C_VEL
LIN {X 0,Y 508.606,Z 944.839,A -85,B 0,C 180,E1 5463.953,E2 5463.953} C_VEL
LIN {X 0,Y 508.08,Z 957.453,A -85,B 0,C 180,E1 5467.207,E2 5467.207} C_VEL
LIN {X 0,Y 507.823,Z 962.995,A -85,B 0,C 180,E1 5469.688,E2 5469.688} C_VEL
LIN {X 0,Y 507.558,Z 965.509,A -85,B 0,C 180,E1 5472.643,E2 5472.643} C_VEL
LIN {X 0,Y 507.766,Z 962.949,A -85,B 0,C 180,E1 5476.199,E2 5476.199} C_VEL
LIN {X 0,Y 508.145,Z 955.604,A -85,B 0,C 180,E1 5479.255,E2 5479.255} C_VEL
LIN {X 0,Y 508.656,Z 942.778,A -85,B 0,C 180,E1 5482.302,E2 5482.302} C_VEL
LIN {X 0,Y 509.515,Z 924.574,A -85,B 0,C 180,E1 5485.098,E2 5485.098} C_VEL
LIN {X 0,Y 510.658,Z 901.809,A -85,B 0,C 180,E1 5487.45,E2 5487.45} C_VEL
LIN {X 0,Y 511.232,Z 875.526,A -85,B 0,C 180,E1 5489.257,E2 5489.257} C_VEL
LIN {X 0,Y 506.719,Z 857.28,A -85,B 0,C 180,E1 5490.353,E2 5490.353} C_VEL
LIN {X 0,Y 507.103,Z 857.28,A -85,B 0,C 180,E1 5495.138,E2 5495.138} C_VEL
LIN {X 0,Y 506.985,Z 857.28,A -85,B 0,C 180,E1 5500.322,E2 5500.322} C_VEL
LIN {X 0,Y 506.818,Z 857.28,A -85,B 0,C 180,E1 5505.596,E2 5505.596} C_VEL
LIN {X 0,Y 506.694,Z 857.28,A -85,B 0,C 180,E1 5511.012,E2 5511.012} C_VEL
LIN {X 0,Y 506.586,Z 857.28,A -85,B 0,C 180,E1 5516.635,E2 5516.635} C_VEL
LIN {X 0,Y 506.454,Z 857.28,A -85,B 0,C 180,E1 5522.555,E2 5522.555} C_VEL
LIN {X 0,Y 506.456,Z 857.28,A -85,B 0,C 180,E1 5526.72,E2 5526.72} C_VEL
LIN {X 0,Y 506.385,Z 857.28,A -85,B 0,C 180,E1 5533.447,E2 5533.447} C_VEL
LIN {X 0,Y 506.463,Z 857.28,A -85,B 0,C 180,E1 5538.927,E2 5538.927} C_VEL
LIN {X 0,Y 506.635,Z 857.28,A -85,B 0,C 180,E1 5540.987,E2 5540.987} C_VEL
LIN {X 0,Y 510.755,Z 880.588,A -85,B 0,C 180,E1 5542.239,E2 5542.239} C_VEL
LIN {X 0,Y 509.968,Z 906.287,A -85,B 0,C 180,E1 5544.101,E2 5544.101} C_VEL
LIN {X 0,Y 509.032,Z 928.206,A -85,B 0,C 180,E1 5546.488,E2 5546.488} C_VEL
LIN {X 0,Y 508.339,Z 945.851,A -85,B 0,C 180,E1 5549.394,E2 5549.394} C_VEL
LIN {X 0,Y 507.993,Z 957.763,A -85,B 0,C 180,E1 5552.524,E2 5552.524} C_VEL
LIN {X 0,Y 507.661,Z 963.615,A -85,B 0,C 180,E1 5555.356,E2 5555.356} C_VEL
LIN {X 0,Y 507.539,Z 965.341,A -85,B 0,C 180,E1 5557.634,E2 5557.634} C_VEL
LIN {X 0,Y 507.783,Z 963.32,A -85,B 0,C 180,E1 5560.885,E2 5560.885} C_VEL
LIN {X 0,Y 508.063,Z 956.192,A -85,B 0,C 180,E1 5564.029,E2 5564.029} C_VEL
LIN {X 0,Y 508.518,Z 943.302,A -85,B 0,C 180,E1 5567.125,E2 5567.125} C_VEL
LIN {X 0,Y 509.206,Z 926.363,A -85,B 0,C 180,E1 5569.75,E2 5569.75} C_VEL
LIN {X 0,Y 510.09,Z 904.675,A -85,B 0,C 180,E1 5572.028,E2 5572.028} C_VEL
LIN {X 0,Y 511.014,Z 879.527,A -85,B 0,C 180,E1 5573.766,E2 5573.766} C_VEL
LIN {X 0,Y 507.184,Z 857.28,A -85,B 0,C 180,E1 5574.993,E2 5574.993} C_VEL
LIN {X 0,Y 507.164,Z 857.28,A -85,B 0,C 180,E1 5580.022,E2 5580.022} C_VEL
LIN {X 0,Y 507.066,Z 857.28,A -85,B 0,C 180,E1 5585.159,E2 5585.159} C_VEL
LIN {X 0,Y 506.967,Z 857.28,A -85,B 0,C 180,E1 5590.34,E2 5590.34} C_VEL
LIN {X 0,Y 506.832,Z 857.28,A -85,B 0,C 180,E1 5595.612,E2 5595.612} C_VEL
LIN {X 0,Y 506.758,Z 857.28,A -85,B 0,C 180,E1 5601.024,E2 5601.024} C_VEL
LIN {X 0,Y 506.621,Z 857.28,A -85,B 0,C 180,E1 5606.646,E2 5606.646} C_VEL
LIN {X 0,Y 506.49,Z 857.28,A -85,B 0,C 180,E1 5612.563,E2 5612.563} C_VEL
LIN {X 0,Y 506.357,Z 857.28,A -85,B 0,C 180,E1 5618.333,E2 5618.333} C_VEL
LIN {X 0,Y 503.883,Z 857.28,A -85,B 0,C 180,E1 5619.793,E2 5619.793} C_VEL
LIN {X 0,Y 498.568,Z 857.28,A -85,B 0,C 180,E1 5621.984,E2 5621.984} C_VEL
LIN {X 0,Y 498.474,Z 857.28,A -85,B 0,C 180,E1 5622.237,E2 5622.237} C_VEL
LIN {X 0,Y 498.574,Z 857.28,A -85,B 0,C 180,E1 5628.08,E2 5628.08} C_VEL
LIN {X 0,Y 498.57,Z 857.28,A -85,B 0,C 180,E1 5634.761,E2 5634.761} C_VEL
LIN {X 0,Y 498.663,Z 857.28,A -85,B 0,C 180,E1 5640.936,E2 5640.936} C_VEL
LIN {X 0,Y 498.769,Z 857.28,A -85,B 0,C 180,E1 5643.203,E2 5643.203} C_VEL
LIN {X 0,Y 508.862,Z 885.947,A -85,B 0,C 180,E1 5644.104,E2 5644.104} C_VEL
LIN {X 0,Y 508.315,Z 939.78,A -85,B 0,C 180,E1 5645.02,E2 5645.02} C_VEL
LIN {X 0,Y 506.98,Z 973.851,A -85,B 0,C 180,E1 5646.243,E2 5646.243} C_VEL
LIN {X 0,Y 505.266,Z 1005.174,A -85,B 0,C 180,E1 5648.084,E2 5648.084} C_VEL
LIN {X 0,Y 503.369,Z 1034.404,A -85,B 0,C 180,E1 5650.565,E2 5650.565} C_VEL
LIN {X 0,Y 501.681,Z 1059.678,A -85,B 0,C 180,E1 5653.565,E2 5653.565} C_VEL
LIN {X 0,Y 500.466,Z 1081.097,A -85,B 0,C 180,E1 5657.108,E2 5657.108} C_VEL
LIN {X 0,Y 499.84,Z 1096.799,A -85,B 0,C 180,E1 5660.893,E2 5660.893} C_VEL
LIN {X 0,Y 499.591,Z 1106.725,A -85,B 0,C 180,E1 5664.784,E2 5664.784} C_VEL
LIN {X 0,Y 499.507,Z 1110.932,A -85,B 0,C 180,E1 5668.264,E2 5668.264} C_VEL
LIN {X 0,Y 499.512,Z 1110.931,A -85,B 0,C 180,E1 5671.738,E2 5671.738} C_VEL
LIN {X 0,Y 499.591,Z 1106.722,A -85,B 0,C 180,E1 5675.217,E2 5675.217} C_VEL
LIN {X 0,Y 499.872,Z 1096.802,A -85,B 0,C 180,E1 5679.106,E2 5679.106} C_VEL
LIN {X 0,Y 500.459,Z 1081.091,A -85,B 0,C 180,E1 5682.893,E2 5682.893} C_VEL
LIN {X 0,Y 501.708,Z 1059.669,A -85,B 0,C 180,E1 5686.435,E2 5686.435} C_VEL
LIN {X 0,Y 503.393,Z 1034.39,A -85,B 0,C 180,E1 5689.435,E2 5689.435} C_VEL
LIN {X 0,Y 505.277,Z 1005.283,A -85,B 0,C 180,E1 5691.907,E2 5691.907} C_VEL
LIN {X 0,Y 506.977,Z 973.113,A -85,B 0,C 180,E1 5693.791,E2 5693.791} C_VEL
LIN {X 0,Y 508.281,Z 938.423,A -85,B 0,C 180,E1 5695.019,E2 5695.019} C_VEL
LIN {X 0,Y 508.287,Z 884.054,A -85,B 0,C 180,E1 5695.945,E2 5695.945} C_VEL
LIN {X 0,Y 498.681,Z 857.28,A -85,B 0,C 180,E1 5696.811,E2 5696.811} C_VEL
LIN {X 0,Y 498.568,Z 857.28,A -85,B 0,C 180,E1 5703.137,E2 5703.137} C_VEL
LIN {X 0,Y 498.441,Z 857.28,A -85,B 0,C 180,E1 5709.636,E2 5709.636} C_VEL
LIN {X 0,Y 498.532,Z 857.28,A -85,B 0,C 180,E1 5715.684,E2 5715.684} C_VEL
LIN {X 0,Y 498.529,Z 857.28,A -85,B 0,C 180,E1 5722.153,E2 5722.153} C_VEL
LIN {X 0,Y 498.538,Z 857.28,A -85,B 0,C 180,E1 5728.253,E2 5728.253} C_VEL
LIN {X 0,Y 498.758,Z 857.28,A -85,B 0,C 180,E1 5734.837,E2 5734.837} C_VEL
LIN {X 0,Y 498.898,Z 857.28,A -85,B 0,C 180,E1 5740.484,E2 5740.484} C_VEL
LIN {X 0,Y 498.798,Z 857.28,A -85,B 0,C 180,E1 5746.253,E2 5746.253} C_VEL
LIN {X 0,Y 499.009,Z 857.28,A -85,B 0,C 180,E1 5751.255,E2 5751.255} C_VEL
LIN {X 0,Y 499.172,Z 857.28,A -85,B 0,C 180,E1 5756.501,E2 5756.501} C_VEL
LIN {X 0,Y 499.185,Z 857.28,A -85,B 0,C 180,E1 5761.715,E2 5761.715} C_VEL
LIN {X 0,Y 499.082,Z 857.28,A -85,B 0,C 180,E1 5766.945,E2 5766.945} C_VEL
LIN {X 0,Y 498.943,Z 857.28,A -85,B 0,C 180,E1 5772.236,E2 5772.236} C_VEL
LIN {X 0,Y 498.894,Z 857.28,A -85,B 0,C 180,E1 5777.636,E2 5777.636} C_VEL
LIN {X 0,Y 498.753,Z 857.28,A -85,B 0,C 180,E1 5783.209,E2 5783.209} C_VEL
LIN {X 0,Y 498.635,Z 857.28,A -85,B 0,C 180,E1 5789.028,E2 5789.028} C_VEL
LIN {X 0,Y 498.524,Z 857.28,A -85,B 0,C 180,E1 5795.199,E2 5795.199} C_VEL
LIN {X 0,Y 498.483,Z 857.28,A -85,B 0,C 180,E1 5801.878,E2 5801.878} C_VEL
LIN {X 0,Y 498.553,Z 857.28,A -85,B 0,C 180,E1 5808.076,E2 5808.076} C_VEL
LIN {X 0,Y 498.802,Z 857.28,A -85,B 0,C 180,E1 5815.132,E2 5815.132} C_VEL
LIN {X 0,Y 504.276,Z 881.807,A -85,B 0,C 180,E1 5816.628,E2 5816.628} C_VEL
LIN {X 0,Y 503.151,Z 906.951,A -85,B 0,C 180,E1 5818.505,E2 5818.505} C_VEL
LIN {X 0,Y 501.866,Z 928.855,A -85,B 0,C 180,E1 5820.943,E2 5820.943} C_VEL
LIN {X 0,Y 500.922,Z 945.887,A -85,B 0,C 180,E1 5823.764,E2 5823.764} C_VEL
LIN {X 0,Y 500.387,Z 957.849,A -85,B 0,C 180,E1 5826.836,E2 5826.836} C_VEL
LIN {X 0,Y 500.044,Z 964.281,A -85,B 0,C 180,E1 5829.694,E2 5829.694} C_VEL
LIN {X 0,Y 499.765,Z 966.636,A -85,B 0,C 180,E1 5832.364,E2 5832.364} C_VEL
LIN {X 0,Y 499.958,Z 964.502,A -85,B 0,C 180,E1 5835.979,E2 5835.979} C_VEL
LIN {X 0,Y 500.344,Z 957.59,A -85,B 0,C 180,E1 5839.085,E2 5839.085} C_VEL
LIN {X 0,Y 500.917,Z 945.338,A -85,B 0,C 180,E1 5842.182,E2 5842.182} C_VEL
LIN {X 0,Y 501.775,Z 927.924,A -85,B 0,C 180,E1 5845.023,E2 5845.023} C_VEL
LIN {X 0,Y 503.062,Z 904.933,A -85,B 0,C 180,E1 5847.52,E2 5847.52} C_VEL
LIN {X 0,Y 504.154,Z 879.533,A -85,B 0,C 180,E1 5849.354,E2 5849.354} C_VEL
LIN {X 0,Y 498.836,Z 857.28,A -85,B 0,C 180,E1 5850.717,E2 5850.717} C_VEL
LIN {X 0,Y 499.195,Z 857.28,A -85,B 0,C 180,E1 5855.22,E2 5855.22} C_VEL
LIN {X 0,Y 499.056,Z 857.28,A -85,B 0,C 180,E1 5860.488,E2 5860.488} C_VEL
LIN {X 0,Y 498.891,Z 857.28,A -85,B 0,C 180,E1 5865.851,E2 5865.851} C_VEL
LIN {X 0,Y 498.763,Z 857.28,A -85,B 0,C 180,E1 5871.363,E2 5871.363} C_VEL
LIN {X 0,Y 498.622,Z 857.28,A -85,B 0,C 180,E1 5877.095,E2 5877.095} C_VEL
LIN {X 0,Y 498.561,Z 857.28,A -85,B 0,C 180,E1 5883.136,E2 5883.136} C_VEL
LIN {X 0,Y 498.405,Z 857.28,A -85,B 0,C 180,E1 5889.638,E2 5889.638} C_VEL
LIN {X 0,Y 498.517,Z 857.28,A -85,B 0,C 180,E1 5895.745,E2 5895.745} C_VEL
LIN {X 0,Y 498.73,Z 858.026,A -85,B 0,C 180,E1 5900.737,E2 5900.737} C_VEL
LIN {X 0,Y 503.182,Z 882.369,A -85,B 0,C 180,E1 5902.063,E2 5902.063} C_VEL
LIN {X 0,Y 502.276,Z 908.737,A -85,B 0,C 180,E1 5904.03,E2 5904.03} C_VEL
LIN {X 0,Y 501.284,Z 930.585,A -85,B 0,C 180,E1 5906.506,E2 5906.506} C_VEL
LIN {X 0,Y 500.598,Z 947.269,A -85,B 0,C 180,E1 5909.338,E2 5909.338} C_VEL
LIN {X 0,Y 500.208,Z 959.371,A -85,B 0,C 180,E1 5912.618,E2 5912.618} C_VEL
LIN {X 0,Y 499.86,Z 964.786,A -85,B 0,C 180,E1 5915.325,E2 5915.325} C_VEL
LIN {X 0,Y 499.762,Z 966.48,A -85,B 0,C 180,E1 5918.715,E2 5918.715} C_VEL
LIN {X 0,Y 500.054,Z 963.633,A -85,B 0,C 180,E1 5921.494,E2 5921.494} C_VEL
LIN {X 0,Y 500.382,Z 955.858,A -85,B 0,C 180,E1 5924.586,E2 5924.586} C_VEL
LIN {X 0,Y 500.948,Z 942.76,A -85,B 0,C 180,E1 5927.592,E2 5927.592} C_VEL
LIN {X 0,Y 501.702,Z 924.929,A -85,B 0,C 180,E1 5930.253,E2 5930.253} C_VEL
LIN {X 0,Y 502.645,Z 901.878,A -85,B 0,C 180,E1 5932.562,E2 5932.562} C_VEL
LIN {X 0,Y 503.182,Z 875.505,A -85,B 0,C 180,E1 5934.284,E2 5934.284} C_VEL
LIN {X 0,Y 499.245,Z 857.28,A -85,B 0,C 180,E1 5935.253,E2 5935.253} C_VEL
LIN {X 0,Y 499.283,Z 857.28,A -85,B 0,C 180,E1 5940.022,E2 5940.022} C_VEL
LIN {X 0,Y 499.172,Z 857.28,A -85,B 0,C 180,E1 5945.241,E2 5945.241} C_VEL
LIN {X 0,Y 499.037,Z 857.28,A -85,B 0,C 180,E1 5950.507,E2 5950.507} C_VEL
LIN {X 0,Y 498.918,Z 857.28,A -85,B 0,C 180,E1 5955.866,E2 5955.866} C_VEL
LIN {X 0,Y 498.853,Z 857.28,A -85,B 0,C 180,E1 5961.373,E2 5961.373} C_VEL
LIN {X 0,Y 498.645,Z 857.28,A -85,B 0,C 180,E1 5967.107,E2 5967.107} C_VEL
LIN {X 0,Y 498.581,Z 857.28,A -85,B 0,C 180,E1 5973.146,E2 5973.146} C_VEL
LIN {X 0,Y 498.443,Z 857.28,A -85,B 0,C 180,E1 5979.644,E2 5979.644} C_VEL
LIN {X 0,Y 498.474,Z 857.28,A -85,B 0,C 180,E1 5982.237,E2 5982.237} C_VEL
LIN {X 0,Y 497.218,Z 857.28,A -85,B 0,C 180,E1 5983.235,E2 5983.235} C_VEL
LIN {X 0,Y 490.676,Z 857.28,A -85,B 0,C 180,E1 5985.955,E2 5985.955} C_VEL
LIN {X 0,Y 490.589,Z 857.28,A -85,B 0,C 180,E1 5986.212,E2 5986.212} C_VEL
LIN {X 0,Y 490.607,Z 857.28,A -85,B 0,C 180,E1 5991.887,E2 5991.887} C_VEL
LIN {X 0,Y 490.681,Z 857.28,A -85,B 0,C 180,E1 5998.362,E2 5998.362} C_VEL
LIN {X 0,Y 490.807,Z 857.28,A -85,B 0,C 180,E1 6002.804,E2 6002.804} C_VEL
LIN {X 0,Y 501.535,Z 888.702,A -85,B 0,C 180,E1 6003.813,E2 6003.813} C_VEL
LIN {X 0,Y 500.886,Z 940.549,A -85,B 0,C 180,E1 6004.73,E2 6004.73} C_VEL
LIN {X 0,Y 499.425,Z 974.654,A -85,B 0,C 180,E1 6005.996,E2 6005.996} C_VEL
LIN {X 0,Y 497.623,Z 1007.694,A -85,B 0,C 180,E1 6007.971,E2 6007.971} C_VEL
LIN {X 0,Y 495.757,Z 1035.495,A -85,B 0,C 180,E1 6010.37,E2 6010.37} C_VEL
LIN {X 0,Y 493.898,Z 1061.276,A -85,B 0,C 180,E1 6013.528,E2 6013.528} C_VEL
LIN {X 0,Y 492.619,Z 1082.182,A -85,B 0,C 180,E1 6017.125,E2 6017.125} C_VEL
LIN {X 0,Y 492.02,Z 1096.092,A -85,B 0,C 180,E1 6020.541,E2 6020.541} C_VEL
LIN {X 0,Y 491.716,Z 1104.992,A -85,B 0,C 180,E1 6023.814,E2 6023.814} C_VEL
LIN {X 0,Y 491.616,Z 1109.407,A -85,B 0,C 180,E1 6026.469,E2 6026.469} C_VEL
LIN {X 0,Y 491.631,Z 1111.5,A -85,B 0,C 180,E1 6030.001,E2 6030.001} C_VEL
LIN {X 0,Y 491.621,Z 1109.404,A -85,B 0,C 180,E1 6033.532,E2 6033.532} C_VEL
LIN {X 0,Y 491.835,Z 1101.849,A -85,B 0,C 180,E1 6037.518,E2 6037.518} C_VEL
LIN {X 0,Y 492.327,Z 1088.281,A -85,B 0,C 180,E1 6041.532,E2 6041.532} C_VEL
LIN {X 0,Y 493.422,Z 1069.134,A -85,B 0,C 180,E1 6045.268,E2 6045.268} C_VEL
LIN {X 0,Y 494.989,Z 1045.523,A -85,B 0,C 180,E1 6048.52,E2 6048.52} C_VEL
LIN {X 0,Y 496.869,Z 1018.394,A -85,B 0,C 180,E1 6051.215,E2 6051.215} C_VEL
LIN {X 0,Y 498.776,Z 987.102,A -85,B 0,C 180,E1 6053.345,E2 6053.345} C_VEL
LIN {X 0,Y 500.384,Z 952.822,A -85,B 0,C 180,E1 6054.889,E2 6054.889} C_VEL
LIN {X 0,Y 501.317,Z 918.387,A -85,B 0,C 180,E1 6055.74,E2 6055.74} C_VEL
LIN {X 0,Y 500.765,Z 885.468,A -85,B 0,C 180,E1 6056.263,E2 6056.263} C_VEL
LIN {X 0,Y 490.751,Z 857.28,A -85,B 0,C 180,E1 6057.227,E2 6057.227} C_VEL
LIN {X 0,Y 490.635,Z 857.28,A -85,B 0,C 180,E1 6063.744,E2 6063.744} C_VEL
LIN {X 0,Y 490.518,Z 857.28,A -85,B 0,C 180,E1 6070.407,E2 6070.407} C_VEL
LIN {X 0,Y 490.605,Z 857.28,A -85,B 0,C 180,E1 6075.221,E2 6075.221} C_VEL
LIN {X 0,Y 490.604,Z 857.28,A -85,B 0,C 180,E1 6080.493,E2 6080.493} C_VEL
LIN {X 0,Y 490.651,Z 857.28,A -85,B 0,C 180,E1 6086.428,E2 6086.428} C_VEL
LIN {X 0,Y 490.715,Z 857.28,A -85,B 0,C 180,E1 6092.418,E2 6092.418} C_VEL
LIN {X 0,Y 490.9,Z 857.28,A -85,B 0,C 180,E1 6098.263,E2 6098.263} C_VEL
LIN {X 0,Y 490.925,Z 857.28,A -85,B 0,C 180,E1 6103.868,E2 6103.868} C_VEL
LIN {X 0,Y 491.041,Z 857.28,A -85,B 0,C 180,E1 6110.645,E2 6110.645} C_VEL
LIN {X 0,Y 491.266,Z 857.28,A -85,B 0,C 180,E1 6116.445,E2 6116.445} C_VEL
LIN {X 0,Y 491.284,Z 857.28,A -85,B 0,C 180,E1 6121.743,E2 6121.743} C_VEL
LIN {X 0,Y 491.17,Z 857.28,A -85,B 0,C 180,E1 6127.057,E2 6127.057} C_VEL
LIN {X 0,Y 491.035,Z 857.28,A -85,B 0,C 180,E1 6132.436,E2 6132.436} C_VEL
LIN {X 0,Y 490.968,Z 857.28,A -85,B 0,C 180,E1 6137.93,E2 6137.93} C_VEL
LIN {X 0,Y 490.826,Z 857.28,A -85,B 0,C 180,E1 6143.606,E2 6143.606} C_VEL
LIN {X 0,Y 490.657,Z 857.28,A -85,B 0,C 180,E1 6149.546,E2 6149.546} C_VEL
LIN {X 0,Y 490.527,Z 857.28,A -85,B 0,C 180,E1 6155.86,E2 6155.86} C_VEL
LIN {X 0,Y 490.576,Z 857.28,A -85,B 0,C 180,E1 6162.206,E2 6162.206} C_VEL
LIN {X 0,Y 490.626,Z 857.28,A -85,B 0,C 180,E1 6167.725,E2 6167.725} C_VEL
LIN {X 0,Y 490.858,Z 857.28,A -85,B 0,C 180,E1 6174.734,E2 6174.734} C_VEL
LIN {X 0,Y 496.91,Z 883.089,A -85,B 0,C 180,E1 6176.341,E2 6176.341} C_VEL
LIN {X 0,Y 495.632,Z 909.219,A -85,B 0,C 180,E1 6178.344,E2 6178.344} C_VEL
LIN {X 0,Y 494.234,Z 931.235,A -85,B 0,C 180,E1 6180.9,E2 6180.9} C_VEL
LIN {X 0,Y 493.179,Z 948.289,A -85,B 0,C 180,E1 6183.858,E2 6183.858} C_VEL
LIN {X 0,Y 492.541,Z 960.22,A -85,B 0,C 180,E1 6187.133,E2 6187.133} C_VEL
LIN {X 0,Y 492.15,Z 966.237,A -85,B 0,C 180,E1 6190.219,E2 6190.219} C_VEL
LIN {X 0,Y 491.955,Z 967.823,A -85,B 0,C 180,E1 6192.415,E2 6192.415} C_VEL
LIN {X 0,Y 492.148,Z 966.04,A -85,B 0,C 180,E1 6195.751,E2 6195.751} C_VEL
LIN {X 0,Y 492.624,Z 958.212,A -85,B 0,C 180,E1 6199.373,E2 6199.373} C_VEL
LIN {X 0,Y 493.251,Z 945.71,A -85,B 0,C 180,E1 6202.503,E2 6202.503} C_VEL
LIN {X 0,Y 494.285,Z 927.572,A -85,B 0,C 180,E1 6205.423,E2 6205.423} C_VEL
LIN {X 0,Y 495.667,Z 904.369,A -85,B 0,C 180,E1 6207.921,E2 6207.921} C_VEL
LIN {X 0,Y 496.482,Z 879.569,A -85,B 0,C 180,E1 6209.715,E2 6209.715} C_VEL
LIN {X 0,Y 490.974,Z 857.28,A -85,B 0,C 180,E1 6211.091,E2 6211.091} C_VEL
LIN {X 0,Y 491.279,Z 857.28,A -85,B 0,C 180,E1 6215.304,E2 6215.304} C_VEL
LIN {X 0,Y 491.131,Z 857.28,A -85,B 0,C 180,E1 6220.659,E2 6220.659} C_VEL
LIN {X 0,Y 490.955,Z 857.28,A -85,B 0,C 180,E1 6226.114,E2 6226.114} C_VEL
LIN {X 0,Y 490.757,Z 857.28,A -85,B 0,C 180,E1 6232.368,E2 6232.368} C_VEL
LIN {X 0,Y 490.709,Z 857.28,A -85,B 0,C 180,E1 6237.569,E2 6237.569} C_VEL
LIN {X 0,Y 490.633,Z 857.28,A -85,B 0,C 180,E1 6243.743,E2 6243.743} C_VEL
LIN {X 0,Y 490.494,Z 857.28,A -85,B 0,C 180,E1 6250.408,E2 6250.408} C_VEL
LIN {X 0,Y 490.586,Z 857.28,A -85,B 0,C 180,E1 6255.221,E2 6255.221} C_VEL
LIN {X 0,Y 490.731,Z 857.617,A -85,B 0,C 180,E1 6260.418,E2 6260.418} C_VEL
LIN {X 0,Y 495.633,Z 882.281,A -85,B 0,C 180,E1 6261.766,E2 6261.766} C_VEL
LIN {X 0,Y 494.791,Z 907.225,A -85,B 0,C 180,E1 6263.596,E2 6263.596} C_VEL
LIN {X 0,Y 493.732,Z 929.072,A -85,B 0,C 180,E1 6265.987,E2 6265.987} C_VEL
LIN {X 0,Y 492.948,Z 946.35,A -85,B 0,C 180,E1 6268.788,E2 6268.788} C_VEL
LIN {X 0,Y 492.445,Z 958.309,A -85,B 0,C 180,E1 6271.774,E2 6271.774} C_VEL
LIN {X 0,Y 492.155,Z 964.817,A -85,B 0,C 180,E1 6274.525,E2 6274.525} C_VEL
LIN {X 0,Y 491.904,Z 967.671,A -85,B 0,C 180,E1 6277.426,E2 6277.426} C_VEL
LIN {X 0,Y 492.226,Z 965.434,A -85,B 0,C 180,E1 6281.189,E2 6281.189} C_VEL
LIN {X 0,Y 492.622,Z 957.319,A -85,B 0,C 180,E1 6284.611,E2 6284.611} C_VEL
LIN {X 0,Y 493.263,Z 943.507,A -85,B 0,C 180,E1 6287.822,E2 6287.822} C_VEL
LIN {X 0,Y 494.141,Z 925.202,A -85,B 0,C 180,E1 6290.547,E2 6290.547} C_VEL
LIN {X 0,Y 495.092,Z 903.031,A -85,B 0,C 180,E1 6292.779,E2 6292.779} C_VEL
LIN {X 0,Y 495.788,Z 877.923,A -85,B 0,C 180,E1 6294.452,E2 6294.452} C_VEL
LIN {X 0,Y 491.321,Z 857.28,A -85,B 0,C 180,E1 6295.606,E2 6295.606} C_VEL
LIN {X 0,Y 491.382,Z 857.28,A -85,B 0,C 180,E1 6300.023,E2 6300.023} C_VEL
LIN {X 0,Y 491.256,Z 857.28,A -85,B 0,C 180,E1 6305.326,E2 6305.326} C_VEL
LIN {X 0,Y 491.118,Z 857.28,A -85,B 0,C 180,E1 6310.678,E2 6310.678} C_VEL
LIN {X 0,Y 490.964,Z 857.28,A -85,B 0,C 180,E1 6317.061,E2 6317.061} C_VEL
LIN {X 0,Y 490.856,Z 857.28,A -85,B 0,C 180,E1 6322.278,E2 6322.278} C_VEL
LIN {X 0,Y 490.703,Z 857.28,A -85,B 0,C 180,E1 6327.582,E2 6327.582} C_VEL
LIN {X 0,Y 490.651,Z 857.28,A -85,B 0,C 180,E1 6333.753,E2 6333.753} C_VEL
LIN {X 0,Y 490.523,Z 857.28,A -85,B 0,C 180,E1 6340.414,E2 6340.414} C_VEL
LIN {X 0,Y 490.589,Z 857.28,A -85,B 0,C 180,E1 6346.212,E2 6346.212} C_VEL
LIN {X 0,Y 488.052,Z 857.28,A -85,B 0,C 180,E1 6347.723,E2 6347.723} C_VEL
LIN {X 0,Y 482.686,Z 857.28,A -85,B 0,C 180,E1 6349.989,E2 6349.989} C_VEL
LIN {X 0,Y 482.599,Z 857.28,A -85,B 0,C 180,E1 6350.251,E2 6350.251} C_VEL
LIN {X 0,Y 482.642,Z 857.28,A -85,B 0,C 180,E1 6355.621,E2 6355.621} C_VEL
LIN {X 0,Y 482.895,Z 857.582,A -85,B 0,C 180,E1 6362.433,E2 6362.433} C_VEL
LIN {X 0,Y 494.201,Z 890.67,A -85,B 0,C 180,E1 6363.5,E2 6363.5} C_VEL
LIN {X 0,Y 493.513,Z 940.414,A -85,B 0,C 180,E1 6364.407,E2 6364.407} C_VEL
LIN {X 0,Y 491.905,Z 974.47,A -85,B 0,C 180,E1 6365.7,E2 6365.7} C_VEL
LIN {X 0,Y 489.961,Z 1007.944,A -85,B 0,C 180,E1 6367.751,E2 6367.751} C_VEL
LIN {X 0,Y 487.869,Z 1037.264,A -85,B 0,C 180,E1 6370.335,E2 6370.335} C_VEL
LIN {X 0,Y 486.216,Z 1061.272,A -85,B 0,C 180,E1 6373.26,E2 6373.26} C_VEL
LIN {X 0,Y 484.82,Z 1082.182,A -85,B 0,C 180,E1 6376.915,E2 6376.915} C_VEL
LIN {X 0,Y 484.164,Z 1096.434,A -85,B 0,C 180,E1 6380.488,E2 6380.488} C_VEL
LIN {X 0,Y 483.789,Z 1106.724,A -85,B 0,C 180,E1 6384.613,E2 6384.613} C_VEL
LIN {X 0,Y 483.732,Z 1110.931,A -85,B 0,C 180,E1 6388.207,E2 6388.207} C_VEL
LIN {X 0,Y 483.736,Z 1110.93,A -85,B 0,C 180,E1 6391.794,E2 6391.794} C_VEL
LIN {X 0,Y 483.79,Z 1106.722,A -85,B 0,C 180,E1 6395.388,E2 6395.388} C_VEL
LIN {X 0,Y 484.175,Z 1096.431,A -85,B 0,C 180,E1 6399.514,E2 6399.514} C_VEL
LIN {X 0,Y 484.947,Z 1080.004,A -85,B 0,C 180,E1 6403.543,E2 6403.543} C_VEL
LIN {X 0,Y 486.331,Z 1059.653,A -85,B 0,C 180,E1 6406.971,E2 6406.971} C_VEL
LIN {X 0,Y 488.085,Z 1034.478,A -85,B 0,C 180,E1 6409.952,E2 6409.952} C_VEL
LIN {X 0,Y 490.187,Z 1004.362,A -85,B 0,C 180,E1 6412.498,E2 6412.498} C_VEL
LIN {X 0,Y 492.036,Z 972.049,A -85,B 0,C 180,E1 6414.402,E2 6414.402} C_VEL
LIN {X 0,Y 493.545,Z 936.822,A -85,B 0,C 180,E1 6415.686,E2 6415.686} C_VEL
LIN {X 0,Y 493.564,Z 887.71,A -85,B 0,C 180,E1 6416.561,E2 6416.561} C_VEL
LIN {X 0,Y 482.808,Z 857.28,A -85,B 0,C 180,E1 6417.653,E2 6417.653} C_VEL
LIN {X 0,Y 482.642,Z 857.28,A -85,B 0,C 180,E1 6424.38,E2 6424.38} C_VEL
LIN {X 0,Y 482.611,Z 857.28,A -85,B 0,C 180,E1 6428.863,E2 6428.863} C_VEL
LIN {X 0,Y 482.585,Z 857.28,A -85,B 0,C 180,E1 6433.805,E2 6433.805} C_VEL
LIN {X 0,Y 482.672,Z 857.28,A -85,B 0,C 180,E1 6438.839,E2 6438.839} C_VEL
LIN {X 0,Y 482.648,Z 857.28,A -85,B 0,C 180,E1 6444.65,E2 6444.65} C_VEL
LIN {X 0,Y 482.735,Z 857.28,A -85,B 0,C 180,E1 6449.866,E2 6449.866} C_VEL
LIN {X 0,Y 482.893,Z 857.28,A -85,B 0,C 180,E1 6455.931,E2 6455.931} C_VEL
LIN {X 0,Y 483.061,Z 857.28,A -85,B 0,C 180,E1 6461.718,E2 6461.718} C_VEL
LIN {X 0,Y 482.985,Z 857.28,A -85,B 0,C 180,E1 6467.306,E2 6467.306} C_VEL
LIN {X 0,Y 483.341,Z 857.28,A -85,B 0,C 180,E1 6472.782,E2 6472.782} C_VEL
LIN {X 0,Y 483.577,Z 857.28,A -85,B 0,C 180,E1 6478.184,E2 6478.184} C_VEL
LIN {X 0,Y 483.501,Z 857.28,A -85,B 0,C 180,E1 6483.566,E2 6483.566} C_VEL
LIN {X 0,Y 483.275,Z 857.28,A -85,B 0,C 180,E1 6488.985,E2 6488.985} C_VEL
LIN {X 0,Y 483.144,Z 857.28,A -85,B 0,C 180,E1 6494.489,E2 6494.489} C_VEL
LIN {X 0,Y 483.026,Z 857.28,A -85,B 0,C 180,E1 6500.136,E2 6500.136} C_VEL
LIN {X 0,Y 482.857,Z 857.28,A -85,B 0,C 180,E1 6506.002,E2 6506.002} C_VEL
LIN {X 0,Y 482.708,Z 857.28,A -85,B 0,C 180,E1 6512.181,E2 6512.181} C_VEL
LIN {X 0,Y 482.611,Z 857.28,A -85,B 0,C 180,E1 6518.813,E2 6518.813} C_VEL
LIN {X 0,Y 482.607,Z 857.28,A -85,B 0,C 180,E1 6523.814,E2 6523.814} C_VEL
LIN {X 0,Y 482.686,Z 857.28,A -85,B 0,C 180,E1 6528.797,E2 6528.797} C_VEL
LIN {X 0,Y 482.872,Z 857.28,A -85,B 0,C 180,E1 6534.301,E2 6534.301} C_VEL
LIN {X 0,Y 489.571,Z 884.319,A -85,B 0,C 180,E1 6536.038,E2 6536.038} C_VEL
LIN {X 0,Y 488.257,Z 909.353,A -85,B 0,C 180,E1 6537.98,E2 6537.98} C_VEL
LIN {X 0,Y 486.729,Z 931.104,A -85,B 0,C 180,E1 6540.485,E2 6540.485} C_VEL
LIN {X 0,Y 485.668,Z 947.486,A -85,B 0,C 180,E1 6543.26,E2 6543.26} C_VEL
LIN {X 0,Y 484.915,Z 959.646,A -85,B 0,C 180,E1 6546.402,E2 6546.402} C_VEL
LIN {X 0,Y 484.399,Z 967.067,A -85,B 0,C 180,E1 6549.889,E2 6549.889} C_VEL
LIN {X 0,Y 484.171,Z 968.936,A -85,B 0,C 180,E1 6553.653,E2 6553.653} C_VEL
LIN {X 0,Y 484.405,Z 966.301,A -85,B 0,C 180,E1 6556.452,E2 6556.452} C_VEL
LIN {X 0,Y 484.919,Z 958.688,A -85,B 0,C 180,E1 6559.704,E2 6559.704} C_VEL
LIN {X 0,Y 485.605,Z 944.849,A -85,B 0,C 180,E1 6563.06,E2 6563.06} C_VEL
LIN {X 0,Y 486.877,Z 926.059,A -85,B 0,C 180,E1 6565.987,E2 6565.987} C_VEL
LIN {X 0,Y 488.361,Z 902.43,A -85,B 0,C 180,E1 6568.445,E2 6568.445} C_VEL
LIN {X 0,Y 488.741,Z 879.741,A -85,B 0,C 180,E1 6570.082,E2 6570.082} C_VEL
LIN {X 0,Y 483.142,Z 857.28,A -85,B 0,C 180,E1 6571.472,E2 6571.472} C_VEL
LIN {X 0,Y 483.295,Z 857.28,A -85,B 0,C 180,E1 6577.198,E2 6577.198} C_VEL
LIN {X 0,Y 483.139,Z 857.28,A -85,B 0,C 180,E1 6582.671,E2 6582.671} C_VEL
LIN {X 0,Y 482.995,Z 857.28,A -85,B 0,C 180,E1 6588.268,E2 6588.268} C_VEL
LIN {X 0,Y 482.773,Z 857.28,A -85,B 0,C 180,E1 6594.673,E2 6594.673} C_VEL
LIN {X 0,Y 482.719,Z 857.28,A -85,B 0,C 180,E1 6600.122,E2 6600.122} C_VEL
LIN {X 0,Y 482.628,Z 857.28,A -85,B 0,C 180,E1 6606.587,E2 6606.587} C_VEL
LIN {X 0,Y 482.578,Z 857.28,A -85,B 0,C 180,E1 6611.213,E2 6611.213} C_VEL
LIN {X 0,Y 482.626,Z 857.28,A -85,B 0,C 180,E1 6616.411,E2 6616.411} C_VEL
LIN {X 0,Y 482.831,Z 857.28,A -85,B 0,C 180,E1 6620.087,E2 6620.087} C_VEL
LIN {X 0,Y 488.076,Z 883.701,A -85,B 0,C 180,E1 6621.557,E2 6621.557} C_VEL
LIN {X 0,Y 487.13,Z 909.625,A -85,B 0,C 180,E1 6623.515,E2 6623.515} C_VEL
LIN {X 0,Y 486.007,Z 931.068,A -85,B 0,C 180,E1 6625.936,E2 6625.936} C_VEL
LIN {X 0,Y 485.167,Z 948.654,A -85,B 0,C 180,E1 6628.909,E2 6628.909} C_VEL
LIN {X 0,Y 484.632,Z 960.634,A -85,B 0,C 180,E1 6632.094,E2 6632.094} C_VEL
LIN {X 0,Y 484.3,Z 966.838,A -85,B 0,C 180,E1 6635.043,E2 6635.043} C_VEL
LIN {X 0,Y 484.108,Z 968.976,A -85,B 0,C 180,E1 6637.991,E2 6637.991} C_VEL
LIN {X 0,Y 484.367,Z 967.138,A -85,B 0,C 180,E1 6640.872,E2 6640.872} C_VEL
LIN {X 0,Y 484.798,Z 960.105,A -85,B 0,C 180,E1 6644.218,E2 6644.218} C_VEL
LIN {X 0,Y 485.406,Z 947.574,A -85,B 0,C 180,E1 6647.417,E2 6647.417} C_VEL
LIN {X 0,Y 486.322,Z 929.16,A -85,B 0,C 180,E1 6650.394,E2 6650.394} C_VEL
LIN {X 0,Y 487.411,Z 906.838,A -85,B 0,C 180,E1 6652.776,E2 6652.776} C_VEL
LIN {X 0,Y 488.412,Z 880.436,A -85,B 0,C 180,E1 6654.616,E2 6654.616} C_VEL
LIN {X 0,Y 483.387,Z 857.28,A -85,B 0,C 180,E1 6655.872,E2 6655.872} C_VEL
LIN {X 0,Y 483.511,Z 857.28,A -85,B 0,C 180,E1 6660.023,E2 6660.023} C_VEL
LIN {X 0,Y 483.354,Z 857.28,A -85,B 0,C 180,E1 6665.413,E2 6665.413} C_VEL
LIN {X 0,Y 483.189,Z 857.28,A -85,B 0,C 180,E1 6670.855,E2 6670.855} C_VEL
LIN {X 0,Y 483.065,Z 857.28,A -85,B 0,C 180,E1 6676.402,E2 6676.402} C_VEL
LIN {X 0,Y 482.98,Z 857.28,A -85,B 0,C 180,E1 6682.112,E2 6682.112} C_VEL
LIN {X 0,Y 482.697,Z 857.28,A -85,B 0,C 180,E1 6688.566,E2 6688.566} C_VEL
LIN {X 0,Y 482.656,Z 857.28,A -85,B 0,C 180,E1 6694.389,E2 6694.389} C_VEL
LIN {X 0,Y 482.614,Z 857.28,A -85,B 0,C 180,E1 6698.872,E2 6698.872} C_VEL
LIN {X 0,Y 482.642,Z 857.28,A -85,B 0,C 180,E1 6703.82,E2 6703.82} C_VEL
LIN {X 0,Y 482.599,Z 857.28,A -85,B 0,C 180,E1 6710.251,E2 6710.251} C_VEL
LIN {X 0,Y 480.079,Z 857.28,A -85,B 0,C 180,E1 6711.786,E2 6711.786} C_VEL
LIN {X 0,Y 474.748,Z 857.28,A -85,B 0,C 180,E1 6714.091,E2 6714.091} C_VEL
LIN {X 0,Y 474.667,Z 857.28,A -85,B 0,C 180,E1 6714.357,E2 6714.357} C_VEL
LIN {X 0,Y 474.834,Z 857.28,A -85,B 0,C 180,E1 6719.426,E2 6719.426} C_VEL
LIN {X 0,Y 474.937,Z 857.831,A -85,B 0,C 180,E1 6722.025,E2 6722.025} C_VEL
LIN {X 0,Y 486.875,Z 892.789,A -85,B 0,C 180,E1 6723.181,E2 6723.181} C_VEL
LIN {X 0,Y 486.17,Z 939.287,A -85,B 0,C 180,E1 6724.045,E2 6724.045} C_VEL
LIN {X 0,Y 484.502,Z 972.886,A -85,B 0,C 180,E1 6725.326,E2 6725.326} C_VEL
LIN {X 0,Y 482.505,Z 1004.769,A -85,B 0,C 180,E1 6727.272,E2 6727.272} C_VEL
LIN {X 0,Y 480.325,Z 1035.202,A -85,B 0,C 180,E1 6729.944,E2 6729.944} C_VEL
LIN {X 0,Y 478.358,Z 1061.842,A -85,B 0,C 180,E1 6733.213,E2 6733.213} C_VEL
LIN {X 0,Y 477.019,Z 1082.12,A -85,B 0,C 180,E1 6736.697,E2 6736.697} C_VEL
LIN {X 0,Y 476.291,Z 1096.705,A -85,B 0,C 180,E1 6740.41,E2 6740.41} C_VEL
LIN {X 0,Y 475.89,Z 1106.724,A -85,B 0,C 180,E1 6744.524,E2 6744.524} C_VEL
LIN {X 0,Y 475.828,Z 1110.931,A -85,B 0,C 180,E1 6748.177,E2 6748.177} C_VEL
LIN {X 0,Y 475.832,Z 1110.93,A -85,B 0,C 180,E1 6751.824,E2 6751.824} C_VEL
LIN {X 0,Y 475.891,Z 1106.721,A -85,B 0,C 180,E1 6755.478,E2 6755.478} C_VEL
LIN {X 0,Y 476.302,Z 1096.68,A -85,B 0,C 180,E1 6759.598,E2 6759.598} C_VEL
LIN {X 0,Y 477.102,Z 1081.001,A -85,B 0,C 180,E1 6763.536,E2 6763.536} C_VEL
LIN {X 0,Y 478.465,Z 1060.13,A -85,B 0,C 180,E1 6767.021,E2 6767.021} C_VEL
LIN {X 0,Y 480.357,Z 1034.115,A -85,B 0,C 180,E1 6770.16,E2 6770.16} C_VEL
LIN {X 0,Y 482.543,Z 1004.54,A -85,B 0,C 180,E1 6772.727,E2 6772.727} C_VEL
LIN {X 0,Y 484.542,Z 972.072,A -85,B 0,C 180,E1 6774.694,E2 6774.694} C_VEL
LIN {X 0,Y 486.142,Z 937.088,A -85,B 0,C 180,E1 6776.004,E2 6776.004} C_VEL
LIN {X 0,Y 486.259,Z 889.709,A -85,B 0,C 180,E1 6776.878,E2 6776.878} C_VEL
LIN {X 0,Y 474.857,Z 857.28,A -85,B 0,C 180,E1 6777.969,E2 6777.969} C_VEL
LIN {X 0,Y 474.708,Z 857.28,A -85,B 0,C 180,E1 6783.971,E2 6783.971} C_VEL
LIN {X 0,Y 474.609,Z 857.28,A -85,B 0,C 180,E1 6790.029,E2 6790.029} C_VEL
LIN {X 0,Y 474.638,Z 857.28,A -85,B 0,C 180,E1 6795.421,E2 6795.421} C_VEL
LIN {X 0,Y 474.688,Z 857.28,A -85,B 0,C 180,E1 6800.353,E2 6800.353} C_VEL
LIN {X 0,Y 474.716,Z 857.28,A -85,B 0,C 180,E1 6806.023,E2 6806.023} C_VEL
LIN {X 0,Y 474.812,Z 857.28,A -85,B 0,C 180,E1 6811.411,E2 6811.411} C_VEL
LIN {X 0,Y 475.037,Z 857.28,A -85,B 0,C 180,E1 6817.566,E2 6817.566} C_VEL
LIN {X 0,Y 475.095,Z 857.28,A -85,B 0,C 180,E1 6823.315,E2 6823.315} C_VEL
LIN {X 0,Y 475.186,Z 857.28,A -85,B 0,C 180,E1 6828.96,E2 6828.96} C_VEL
LIN {X 0,Y 475.477,Z 857.28,A -85,B 0,C 180,E1 6834.497,E2 6834.497} C_VEL
LIN {X 0,Y 475.628,Z 857.28,A -85,B 0,C 180,E1 6839.977,E2 6839.977} C_VEL
LIN {X 0,Y 475.429,Z 857.28,A -85,B 0,C 180,E1 6845.457,E2 6845.457} C_VEL
LIN {X 0,Y 475.255,Z 857.28,A -85,B 0,C 180,E1 6850.991,E2 6850.991} C_VEL
LIN {X 0,Y 475.122,Z 857.28,A -85,B 0,C 180,E1 6857.055,E2 6857.055} C_VEL
LIN {X 0,Y 475.002,Z 857.28,A -85,B 0,C 180,E1 6862.453,E2 6862.453} C_VEL
LIN {X 0,Y 474.845,Z 857.28,A -85,B 0,C 180,E1 6868.533,E2 6868.533} C_VEL
LIN {X 0,Y 474.693,Z 857.28,A -85,B 0,C 180,E1 6874.993,E2 6874.993} C_VEL
LIN {X 0,Y 474.599,Z 857.28,A -85,B 0,C 180,E1 6882.009,E2 6882.009} C_VEL
LIN {X 0,Y 474.696,Z 857.28,A -85,B 0,C 180,E1 6887.947,E2 6887.947} C_VEL
LIN {X 0,Y 474.924,Z 857.744,A -85,B 0,C 180,E1 6893.872,E2 6893.872} C_VEL
LIN {X 0,Y 482.239,Z 885.273,A -85,B 0,C 180,E1 6895.704,E2 6895.704} C_VEL
LIN {X 0,Y 480.841,Z 909.899,A -85,B 0,C 180,E1 6897.635,E2 6897.635} C_VEL
LIN {X 0,Y 479.249,Z 931.46,A -85,B 0,C 180,E1 6900.131,E2 6900.131} C_VEL
LIN {X 0,Y 478.032,Z 948.298,A -85,B 0,C 180,E1 6902.996,E2 6902.996} C_VEL
LIN {X 0,Y 477.167,Z 960.974,A -85,B 0,C 180,E1 6906.327,E2 6906.327} C_VEL
LIN {X 0,Y 476.645,Z 967.901,A -85,B 0,C 180,E1 6909.548,E2 6909.548} C_VEL
LIN {X 0,Y 476.358,Z 970.169,A -85,B 0,C 180,E1 6913.377,E2 6913.377} C_VEL
LIN {X 0,Y 476.678,Z 966.387,A -85,B 0,C 180,E1 6917.153,E2 6917.153} C_VEL
LIN {X 0,Y 477.273,Z 957.598,A -85,B 0,C 180,E1 6920.511,E2 6920.511} C_VEL
LIN {X 0,Y 478.24,Z 942.615,A -85,B 0,C 180,E1 6923.866,E2 6923.866} C_VEL
LIN {X 0,Y 479.568,Z 924.024,A -85,B 0,C 180,E1 6926.606,E2 6926.606} C_VEL
LIN {X 0,Y 481.101,Z 900.29,A -85,B 0,C 180,E1 6928.985,E2 6928.985} C_VEL
LIN {X 0,Y 481.162,Z 880.957,A -85,B 0,C 180,E1 6930.379,E2 6930.379} C_VEL
LIN {X 0,Y 475.312,Z 857.28,A -85,B 0,C 180,E1 6931.939,E2 6931.939} C_VEL
LIN {X 0,Y 475.378,Z 857.28,A -85,B 0,C 180,E1 6937.319,E2 6937.319} C_VEL
LIN {X 0,Y 475.223,Z 857.28,A -85,B 0,C 180,E1 6942.886,E2 6942.886} C_VEL
LIN {X 0,Y 475.079,Z 857.28,A -85,B 0,C 180,E1 6948.584,E2 6948.584} C_VEL
LIN {X 0,Y 474.878,Z 857.28,A -85,B 0,C 180,E1 6954.486,E2 6954.486} C_VEL
LIN {X 0,Y 474.774,Z 857.28,A -85,B 0,C 180,E1 6960.68,E2 6960.68} C_VEL
LIN {X 0,Y 474.681,Z 857.28,A -85,B 0,C 180,E1 6967.303,E2 6967.303} C_VEL
LIN {X 0,Y 474.604,Z 857.28,A -85,B 0,C 180,E1 6972.86,E2 6972.86} C_VEL
LIN {X 0,Y 474.924,Z 857.445,A -85,B 0,C 180,E1 6979.792,E2 6979.792} C_VEL
LIN {X 0,Y 480.534,Z 884.305,A -85,B 0,C 180,E1 6981.291,E2 6981.291} C_VEL
LIN {X 0,Y 479.565,Z 909.446,A -85,B 0,C 180,E1 6983.187,E2 6983.187} C_VEL
LIN {X 0,Y 478.354,Z 931.716,A -85,B 0,C 180,E1 6985.702,E2 6985.702} C_VEL
LIN {X 0,Y 477.46,Z 949.041,A -85,B 0,C 180,E1 6988.621,E2 6988.621} C_VEL
LIN {X 0,Y 476.885,Z 960.599,A -85,B 0,C 180,E1 6991.6,E2 6991.6} C_VEL
LIN {X 0,Y 476.554,Z 967.451,A -85,B 0,C 180,E1 6994.609,E2 6994.609} C_VEL
LIN {X 0,Y 476.299,Z 970.098,A -85,B 0,C 180,E1 6997.611,E2 6997.611} C_VEL
LIN {X 0,Y 476.546,Z 968.802,A -85,B 0,C 180,E1 7000.546,E2 7000.546} C_VEL
LIN {X 0,Y 476.964,Z 962.464,A -85,B 0,C 180,E1 7003.905,E2 7003.905} C_VEL
LIN {X 0,Y 477.616,Z 950.499,A -85,B 0,C 180,E1 7007.209,E2 7007.209} C_VEL
LIN {X 0,Y 478.574,Z 932.907,A -85,B 0,C 180,E1 7010.237,E2 7010.237} C_VEL
LIN {X 0,Y 479.715,Z 910.64,A -85,B 0,C 180,E1 7012.774,E2 7012.774} C_VEL
LIN {X 0,Y 480.853,Z 885.136,A -85,B 0,C 180,E1 7014.668,E2 7014.668} C_VEL
LIN {X 0,Y 476.499,Z 862.111,A -85,B 0,C 180,E1 7015.962,E2 7015.962} C_VEL
LIN {X 0,Y 475.474,Z 857.28,A -85,B 0,C 180,E1 7016.221,E2 7016.221} C_VEL
LIN {X 0,Y 475.499,Z 857.28,A -85,B 0,C 180,E1 7021.847,E2 7021.847} C_VEL
LIN {X 0,Y 475.349,Z 857.28,A -85,B 0,C 180,E1 7027.34,E2 7027.34} C_VEL
LIN {X 0,Y 475.202,Z 857.28,A -85,B 0,C 180,E1 7032.905,E2 7032.905} C_VEL
LIN {X 0,Y 475.106,Z 857.28,A -85,B 0,C 180,E1 7038.6,E2 7038.6} C_VEL
LIN {X 0,Y 474.987,Z 857.28,A -85,B 0,C 180,E1 7044.495,E2 7044.495} C_VEL
LIN {X 0,Y 474.794,Z 857.28,A -85,B 0,C 180,E1 7050.691,E2 7050.691} C_VEL
LIN {X 0,Y 474.696,Z 857.28,A -85,B 0,C 180,E1 7057.313,E2 7057.313} C_VEL
LIN {X 0,Y 474.635,Z 857.28,A -85,B 0,C 180,E1 7062.804,E2 7062.804} C_VEL
LIN {X 0,Y 474.705,Z 857.28,A -85,B 0,C 180,E1 7067.949,E2 7067.949} C_VEL
LIN {X 0,Y 474.667,Z 857.28,A -85,B 0,C 180,E1 7074.357,E2 7074.357} C_VEL
LIN {X 0,Y 472.172,Z 857.28,A -85,B 0,C 180,E1 7075.916,E2 7075.916} C_VEL
LIN {X 0,Y 466.887,Z 857.28,A -85,B 0,C 180,E1 7078.258,E2 7078.258} C_VEL
LIN {X 0,Y 466.815,Z 857.28,A -85,B 0,C 180,E1 7078.528,E2 7078.528} C_VEL
LIN {X 0,Y 466.976,Z 857.28,A -85,B 0,C 180,E1 7081.55,E2 7081.55} C_VEL
LIN {X 0,Y 479.497,Z 892.783,A -85,B 0,C 180,E1 7082.815,E2 7082.815} C_VEL
LIN {X 0,Y 478.853,Z 938.228,A -85,B 0,C 180,E1 7083.674,E2 7083.674} C_VEL
LIN {X 0,Y 477.033,Z 972.247,A -85,B 0,C 180,E1 7084.987,E2 7084.987} C_VEL
LIN {X 0,Y 474.882,Z 1004.693,A -85,B 0,C 180,E1 7087.011,E2 7087.011} C_VEL
LIN {X 0,Y 472.595,Z 1034.926,A -85,B 0,C 180,E1 7089.733,E2 7089.733} C_VEL
LIN {X 0,Y 470.597,Z 1060.494,A -85,B 0,C 180,E1 7092.928,E2 7092.928} C_VEL
LIN {X 0,Y 469.195,Z 1081.215,A -85,B 0,C 180,E1 7096.525,E2 7096.525} C_VEL
LIN {X 0,Y 468.396,Z 1096.774,A -85,B 0,C 180,E1 7100.367,E2 7100.367} C_VEL
LIN {X 0,Y 467.992,Z 1106.722,A -85,B 0,C 180,E1 7104.431,E2 7104.431} C_VEL
LIN {X 0,Y 467.938,Z 1110.931,A -85,B 0,C 180,E1 7108.146,E2 7108.146} C_VEL
LIN {X 0,Y 467.942,Z 1110.929,A -85,B 0,C 180,E1 7111.855,E2 7111.855} C_VEL
LIN {X 0,Y 467.992,Z 1106.72,A -85,B 0,C 180,E1 7115.57,E2 7115.57} C_VEL
LIN {X 0,Y 468.406,Z 1096.771,A -85,B 0,C 180,E1 7119.635,E2 7119.635} C_VEL
LIN {X 0,Y 469.185,Z 1081.212,A -85,B 0,C 180,E1 7123.469,E2 7123.469} C_VEL
LIN {X 0,Y 470.608,Z 1060.392,A -85,B 0,C 180,E1 7127.073,E2 7127.073} C_VEL
LIN {X 0,Y 472.652,Z 1033.621,A -85,B 0,C 180,E1 7130.388,E2 7130.388} C_VEL
LIN {X 0,Y 474.919,Z 1004.366,A -85,B 0,C 180,E1 7132.989,E2 7132.989} C_VEL
LIN {X 0,Y 477.115,Z 971.268,A -85,B 0,C 180,E1 7135.034,E2 7135.034} C_VEL
LIN {X 0,Y 478.818,Z 936.128,A -85,B 0,C 180,E1 7136.367,E2 7136.367} C_VEL
LIN {X 0,Y 479.005,Z 891.61,A -85,B 0,C 180,E1 7137.204,E2 7137.204} C_VEL
LIN {X 0,Y 466.941,Z 857.28,A -85,B 0,C 180,E1 7138.435,E2 7138.435} C_VEL
LIN {X 0,Y 466.799,Z 857.28,A -85,B 0,C 180,E1 7143.464,E2 7143.464} C_VEL
LIN {X 0,Y 466.671,Z 857.28,A -85,B 0,C 180,E1 7150.458,E2 7150.458} C_VEL
LIN {X 0,Y 466.773,Z 857.28,A -85,B 0,C 180,E1 7157.055,E2 7157.055} C_VEL
LIN {X 0,Y 466.75,Z 857.28,A -85,B 0,C 180,E1 7161.94,E2 7161.94} C_VEL
LIN {X 0,Y 466.805,Z 857.28,A -85,B 0,C 180,E1 7168.725,E2 7168.725} C_VEL
LIN {X 0,Y 467.038,Z 857.28,A -85,B 0,C 180,E1 7175.194,E2 7175.194} C_VEL
LIN {X 0,Y 467.188,Z 857.28,A -85,B 0,C 180,E1 7181.073,E2 7181.073} C_VEL
LIN {X 0,Y 467.137,Z 857.28,A -85,B 0,C 180,E1 7186.868,E2 7186.868} C_VEL
LIN {X 0,Y 467.489,Z 857.28,A -85,B 0,C 180,E1 7192.536,E2 7192.536} C_VEL
LIN {X 0,Y 467.769,Z 857.28,A -85,B 0,C 180,E1 7198.122,E2 7198.122} C_VEL
LIN {X 0,Y 467.702,Z 857.28,A -85,B 0,C 180,E1 7203.687,E2 7203.687} C_VEL
LIN {X 0,Y 467.433,Z 857.28,A -85,B 0,C 180,E1 7209.292,E2 7209.292} C_VEL
LIN {X 0,Y 467.264,Z 857.28,A -85,B 0,C 180,E1 7214.993,E2 7214.993} C_VEL
LIN {X 0,Y 467.121,Z 857.28,A -85,B 0,C 180,E1 7220.853,E2 7220.853} C_VEL
LIN {X 0,Y 466.941,Z 857.28,A -85,B 0,C 180,E1 7226.958,E2 7226.958} C_VEL
LIN {X 0,Y 466.767,Z 857.28,A -85,B 0,C 180,E1 7233.421,E2 7233.421} C_VEL
LIN {X 0,Y 466.667,Z 857.28,A -85,B 0,C 180,E1 7240.405,E2 7240.405} C_VEL
LIN {X 0,Y 466.774,Z 857.28,A -85,B 0,C 180,E1 7247.063,E2 7247.063} C_VEL
LIN {X 0,Y 467.014,Z 858.072,A -85,B 0,C 180,E1 7253.415,E2 7253.415} C_VEL
LIN {X 0,Y 474.722,Z 885.759,A -85,B 0,C 180,E1 7255.312,E2 7255.312} C_VEL
LIN {X 0,Y 473.421,Z 911.529,A -85,B 0,C 180,E1 7257.383,E2 7257.383} C_VEL
LIN {X 0,Y 471.647,Z 933.42,A -85,B 0,C 180,E1 7259.993,E2 7259.993} C_VEL
LIN {X 0,Y 470.214,Z 951.322,A -85,B 0,C 180,E1 7263.204,E2 7263.204} C_VEL
LIN {X 0,Y 469.371,Z 962.918,A -85,B 0,C 180,E1 7266.469,E2 7266.469} C_VEL
LIN {X 0,Y 468.876,Z 968.875,A -85,B 0,C 180,E1 7269.332,E2 7269.332} C_VEL
LIN {X 0,Y 468.541,Z 971.408,A -85,B 0,C 180,E1 7273.092,E2 7273.092} C_VEL
LIN {X 0,Y 468.867,Z 968.021,A -85,B 0,C 180,E1 7276.935,E2 7276.935} C_VEL
LIN {X 0,Y 469.499,Z 959.487,A -85,B 0,C 180,E1 7280.409,E2 7280.409} C_VEL
LIN {X 0,Y 470.478,Z 945.339,A -85,B 0,C 180,E1 7283.764,E2 7283.764} C_VEL
LIN {X 0,Y 471.953,Z 925.646,A -85,B 0,C 180,E1 7286.781,E2 7286.781} C_VEL
LIN {X 0,Y 473.601,Z 902.168,A -85,B 0,C 180,E1 7289.198,E2 7289.198} C_VEL
LIN {X 0,Y 473.954,Z 883.838,A -85,B 0,C 180,E1 7290.559,E2 7290.559} C_VEL
LIN {X 0,Y 467.447,Z 857.28,A -85,B 0,C 180,E1 7292.271,E2 7292.271} C_VEL
LIN {X 0,Y 467.49,Z 857.28,A -85,B 0,C 180,E1 7297.443,E2 7297.443} C_VEL
LIN {X 0,Y 467.257,Z 857.28,A -85,B 0,C 180,E1 7303.767,E2 7303.767} C_VEL
LIN {X 0,Y 467.092,Z 857.28,A -85,B 0,C 180,E1 7310.08,E2 7310.08} C_VEL
LIN {X 0,Y 466.935,Z 857.28,A -85,B 0,C 180,E1 7314.931,E2 7314.931} C_VEL
LIN {X 0,Y 466.787,Z 857.28,A -85,B 0,C 180,E1 7321.263,E2 7321.263} C_VEL
LIN {X 0,Y 466.665,Z 857.28,A -85,B 0,C 180,E1 7328.056,E2 7328.056} C_VEL
LIN {X 0,Y 466.725,Z 857.28,A -85,B 0,C 180,E1 7334.523,E2 7334.523} C_VEL
LIN {X 0,Y 466.975,Z 857.733,A -85,B 0,C 180,E1 7339.483,E2 7339.483} C_VEL
LIN {X 0,Y 472.864,Z 884.659,A -85,B 0,C 180,E1 7340.997,E2 7340.997} C_VEL
LIN {X 0,Y 471.956,Z 910.869,A -85,B 0,C 180,E1 7343.004,E2 7343.004} C_VEL
LIN {X 0,Y 470.667,Z 933.038,A -85,B 0,C 180,E1 7345.553,E2 7345.553} C_VEL
LIN {X 0,Y 469.752,Z 949.481,A -85,B 0,C 180,E1 7348.34,E2 7348.34} C_VEL
LIN {X 0,Y 469.104,Z 962.221,A -85,B 0,C 180,E1 7351.679,E2 7351.679} C_VEL
LIN {X 0,Y 468.689,Z 969.504,A -85,B 0,C 180,E1 7355.206,E2 7355.206} C_VEL
LIN {X 0,Y 468.523,Z 971.18,A -85,B 0,C 180,E1 7357.219,E2 7357.219} C_VEL
LIN {X 0,Y 468.654,Z 970.917,A -85,B 0,C 180,E1 7359.536,E2 7359.536} C_VEL
LIN {X 0,Y 469.074,Z 965.787,A -85,B 0,C 180,E1 7363.144,E2 7363.144} C_VEL
LIN {X 0,Y 469.677,Z 955.066,A -85,B 0,C 180,E1 7366.586,E2 7366.586} C_VEL
LIN {X 0,Y 470.654,Z 939.014,A -85,B 0,C 180,E1 7369.708,E2 7369.708} C_VEL
LIN {X 0,Y 471.937,Z 917.732,A -85,B 0,C 180,E1 7372.422,E2 7372.422} C_VEL
LIN {X 0,Y 473.079,Z 892.869,A -85,B 0,C 180,E1 7374.516,E2 7374.516} C_VEL
LIN {X 0,Y 472.557,Z 878.91,A -85,B 0,C 180,E1 7375.385,E2 7375.385} C_VEL
LIN {X 0,Y 467.571,Z 857.28,A -85,B 0,C 180,E1 7376.544,E2 7376.544} C_VEL
LIN {X 0,Y 467.628,Z 857.28,A -85,B 0,C 180,E1 7381.878,E2 7381.878} C_VEL
LIN {X 0,Y 467.435,Z 857.28,A -85,B 0,C 180,E1 7387.465,E2 7387.465} C_VEL
LIN {X 0,Y 467.239,Z 857.28,A -85,B 0,C 180,E1 7393.558,E2 7393.558} C_VEL
LIN {X 0,Y 467.135,Z 857.28,A -85,B 0,C 180,E1 7399.959,E2 7399.959} C_VEL
LIN {X 0,Y 467.017,Z 857.28,A -85,B 0,C 180,E1 7404.942,E2 7404.942} C_VEL
LIN {X 0,Y 466.818,Z 857.28,A -85,B 0,C 180,E1 7411.274,E2 7411.274} C_VEL
LIN {X 0,Y 466.687,Z 857.28,A -85,B 0,C 180,E1 7418.066,E2 7418.066} C_VEL
LIN {X 0,Y 466.76,Z 857.28,A -85,B 0,C 180,E1 7424.469,E2 7424.469} C_VEL
LIN {X 0,Y 466.765,Z 857.28,A -85,B 0,C 180,E1 7429.553,E2 7429.553} C_VEL
LIN {X 0,Y 466.798,Z 857.28,A -85,B 0,C 180,E1 7436.538,E2 7436.538} C_VEL
LIN {X 0,Y 466.815,Z 857.28,A -85,B 0,C 180,E1 7438.528,E2 7438.528} C_VEL
LIN {X 0,Y 462.872,Z 857.28,A -85,B 0,C 180,E1 7439.383,E2 7439.383} C_VEL
LIN {X 0,Y 458.915,Z 857.28,A -85,B 0,C 180,E1 7440.253,E2 7440.253} C_VEL
LIN {X 0,Y 459.032,Z 857.28,A -85,B 0,C 180,E1 7441.148,E2 7441.148} C_VEL
LIN {X 0,Y 472.331,Z 896,A -85,B 0,C 180,E1 7442.499,E2 7442.499} C_VEL
LIN {X 0,Y 471.492,Z 938.449,A -85,B 0,C 180,E1 7443.33,E2 7443.33} C_VEL
LIN {X 0,Y 469.511,Z 973.278,A -85,B 0,C 180,E1 7444.73,E2 7444.73} C_VEL
LIN {X 0,Y 467.151,Z 1006.209,A -85,B 0,C 180,E1 7446.861,E2 7446.861} C_VEL
LIN {X 0,Y 464.758,Z 1035.653,A -85,B 0,C 180,E1 7449.625,E2 7449.625} C_VEL
LIN {X 0,Y 462.711,Z 1060.714,A -85,B 0,C 180,E1 7452.873,E2 7452.873} C_VEL
LIN {X 0,Y 461.241,Z 1081.973,A -85,B 0,C 180,E1 7456.716,E2 7456.716} C_VEL
LIN {X 0,Y 460.507,Z 1096.589,A -85,B 0,C 180,E1 7460.539,E2 7460.539} C_VEL
LIN {X 0,Y 460.149,Z 1105.835,A -85,B 0,C 180,E1 7464.336,E2 7464.336} C_VEL
LIN {X 0,Y 460.054,Z 1110.336,A -85,B 0,C 180,E1 7468.115,E2 7468.115} C_VEL
LIN {X 0,Y 460.057,Z 1110.334,A -85,B 0,C 180,E1 7471.887,E2 7471.887} C_VEL
LIN {X 0,Y 460.149,Z 1105.823,A -85,B 0,C 180,E1 7475.666,E2 7475.666} C_VEL
LIN {X 0,Y 460.564,Z 1095.206,A -85,B 0,C 180,E1 7479.891,E2 7479.891} C_VEL
LIN {X 0,Y 461.46,Z 1078.27,A -85,B 0,C 180,E1 7484.04,E2 7484.04} C_VEL
LIN {X 0,Y 463.004,Z 1056.535,A -85,B 0,C 180,E1 7487.716,E2 7487.716} C_VEL
LIN {X 0,Y 465.2,Z 1029.772,A -85,B 0,C 180,E1 7490.979,E2 7490.979} C_VEL
LIN {X 0,Y 467.627,Z 999.383,A -85,B 0,C 180,E1 7493.621,E2 7493.621} C_VEL
LIN {X 0,Y 469.878,Z 967.109,A -85,B 0,C 180,E1 7495.544,E2 7495.544} C_VEL
LIN {X 0,Y 471.632,Z 932.561,A -85,B 0,C 180,E1 7496.812,E2 7496.812} C_VEL
LIN {X 0,Y 471.522,Z 893.121,A -85,B 0,C 180,E1 7497.56,E2 7497.56} C_VEL
LIN {X 0,Y 458.982,Z 857.28,A -85,B 0,C 180,E1 7498.851,E2 7498.851} C_VEL
LIN {X 0,Y 458.806,Z 857.28,A -85,B 0,C 180,E1 7504.404,E2 7504.404} C_VEL
LIN {X 0,Y 458.758,Z 857.28,A -85,B 0,C 180,E1 7510.608,E2 7510.608} C_VEL
LIN {X 0,Y 458.843,Z 857.28,A -85,B 0,C 180,E1 7516.549,E2 7516.549} C_VEL
LIN {X 0,Y 458.821,Z 857.28,A -85,B 0,C 180,E1 7522.372,E2 7522.372} C_VEL
LIN {X 0,Y 458.889,Z 857.28,A -85,B 0,C 180,E1 7529.078,E2 7529.078} C_VEL
LIN {X 0,Y 459.051,Z 857.28,A -85,B 0,C 180,E1 7534.595,E2 7534.595} C_VEL
LIN {X 0,Y 459.282,Z 857.28,A -85,B 0,C 180,E1 7540.735,E2 7540.735} C_VEL
LIN {X 0,Y 459.227,Z 857.28,A -85,B 0,C 180,E1 7546.637,E2 7546.637} C_VEL
LIN {X 0,Y 459.56,Z 857.28,A -85,B 0,C 180,E1 7552.406,E2 7552.406} C_VEL
LIN {X 0,Y 459.859,Z 857.28,A -85,B 0,C 180,E1 7558.09,E2 7558.09} C_VEL
LIN {X 0,Y 459.785,Z 857.28,A -85,B 0,C 180,E1 7563.75,E2 7563.75} C_VEL
LIN {X 0,Y 459.518,Z 857.28,A -85,B 0,C 180,E1 7569.454,E2 7569.454} C_VEL
LIN {X 0,Y 459.329,Z 857.28,A -85,B 0,C 180,E1 7575.258,E2 7575.258} C_VEL
LIN {X 0,Y 459.163,Z 857.28,A -85,B 0,C 180,E1 7581.232,E2 7581.232} C_VEL
LIN {X 0,Y 458.999,Z 857.28,A -85,B 0,C 180,E1 7587.464,E2 7587.464} C_VEL
LIN {X 0,Y 458.779,Z 857.28,A -85,B 0,C 180,E1 7594.082,E2 7594.082} C_VEL
LIN {X 0,Y 458.772,Z 857.28,A -85,B 0,C 180,E1 7600.617,E2 7600.617} C_VEL
LIN {X 0,Y 458.831,Z 857.28,A -85,B 0,C 180,E1 7606.488,E2 7606.488} C_VEL
LIN {X 0,Y 459.063,Z 857.88,A -85,B 0,C 180,E1 7612.911,E2 7612.911} C_VEL
LIN {X 0,Y 466.947,Z 885.669,A -85,B 0,C 180,E1 7614.849,E2 7614.849} C_VEL
LIN {X 0,Y 466.555,Z 905.426,A -85,B 0,C 180,E1 7616.39,E2 7616.39} C_VEL
LIN {X 0,Y 464.732,Z 928.24,A -85,B 0,C 180,E1 7618.852,E2 7618.852} C_VEL
LIN {X 0,Y 463.088,Z 947.216,A -85,B 0,C 180,E1 7621.881,E2 7621.881} C_VEL
LIN {X 0,Y 461.872,Z 961.023,A -85,B 0,C 180,E1 7625.271,E2 7625.271} C_VEL
LIN {X 0,Y 461.167,Z 969.404,A -85,B 0,C 180,E1 7628.829,E2 7628.829} C_VEL
LIN {X 0,Y 460.74,Z 972.592,A -85,B 0,C 180,E1 7632.796,E2 7632.796} C_VEL
LIN {X 0,Y 461.025,Z 969.658,A -85,B 0,C 180,E1 7636.709,E2 7636.709} C_VEL
LIN {X 0,Y 461.666,Z 962.201,A -85,B 0,C 180,E1 7640.04,E2 7640.04} C_VEL
LIN {X 0,Y 462.494,Z 949.148,A -85,B 0,C 180,E1 7643.42,E2 7643.42} C_VEL
LIN {X 0,Y 464.031,Z 930.792,A -85,B 0,C 180,E1 7646.492,E2 7646.492} C_VEL
LIN {X 0,Y 465.771,Z 907.979,A -85,B 0,C 180,E1 7649.068,E2 7649.068} C_VEL
LIN {X 0,Y 466.446,Z 885.235,A -85,B 0,C 180,E1 7650.853,E2 7650.853} C_VEL
LIN {X 0,Y 459.593,Z 857.28,A -85,B 0,C 180,E1 7652.714,E2 7652.714} C_VEL
LIN {X 0,Y 459.527,Z 857.28,A -85,B 0,C 180,E1 7659.03,E2 7659.03} C_VEL
LIN {X 0,Y 459.32,Z 857.28,A -85,B 0,C 180,E1 7665.289,E2 7665.289} C_VEL
LIN {X 0,Y 459.113,Z 857.28,A -85,B 0,C 180,E1 7671.269,E2 7671.269} C_VEL
LIN {X 0,Y 458.951,Z 857.28,A -85,B 0,C 180,E1 7677.506,E2 7677.506} C_VEL
LIN {X 0,Y 458.792,Z 857.28,A -85,B 0,C 180,E1 7684.126,E2 7684.126} C_VEL
LIN {X 0,Y 458.744,Z 857.28,A -85,B 0,C 180,E1 7690.68,E2 7690.68} C_VEL
LIN {X 0,Y 458.831,Z 857.28,A -85,B 0,C 180,E1 7696.549,E2 7696.549} C_VEL
LIN {X 0,Y 459.031,Z 857.339,A -85,B 0,C 180,E1 7699.139,E2 7699.139} C_VEL
LIN {X 0,Y 465.139,Z 885.04,A -85,B 0,C 180,E1 7700.702,E2 7700.702} C_VEL
LIN {X 0,Y 464.403,Z 911.001,A -85,B 0,C 180,E1 7702.695,E2 7702.695} C_VEL
LIN {X 0,Y 463.009,Z 933.845,A -85,B 0,C 180,E1 7705.333,E2 7705.333} C_VEL
LIN {X 0,Y 461.952,Z 951.731,A -85,B 0,C 180,E1 7708.447,E2 7708.447} C_VEL
LIN {X 0,Y 461.298,Z 964.6,A -85,B 0,C 180,E1 7712.03,E2 7712.03} C_VEL
LIN {X 0,Y 460.926,Z 970.129,A -85,B 0,C 180,E1 7714.759,E2 7714.759} C_VEL
LIN {X 0,Y 460.742,Z 972.244,A -85,B 0,C 180,E1 7716.943,E2 7716.943} C_VEL
LIN {X 0,Y 460.779,Z 972.451,A -85,B 0,C 180,E1 7718.846,E2 7718.846} C_VEL
LIN {X 0,Y 461.203,Z 969.099,A -85,B 0,C 180,E1 7722.18,E2 7722.18} C_VEL
LIN {X 0,Y 461.745,Z 960.227,A -85,B 0,C 180,E1 7725.667,E2 7725.667} C_VEL
LIN {X 0,Y 462.764,Z 945.692,A -85,B 0,C 180,E1 7728.971,E2 7728.971} C_VEL
LIN {X 0,Y 463.913,Z 926.382,A -85,B 0,C 180,E1 7731.819,E2 7731.819} C_VEL
LIN {X 0,Y 465.212,Z 902.823,A -85,B 0,C 180,E1 7734.138,E2 7734.138} C_VEL
LIN {X 0,Y 465.433,Z 882.145,A -85,B 0,C 180,E1 7735.541,E2 7735.541} C_VEL
LIN {X 0,Y 459.7,Z 857.28,A -85,B 0,C 180,E1 7736.957,E2 7736.957} C_VEL
LIN {X 0,Y 459.726,Z 857.28,A -85,B 0,C 180,E1 7741.911,E2 7741.911} C_VEL
LIN {X 0,Y 459.499,Z 857.28,A -85,B 0,C 180,E1 7748.695,E2 7748.695} C_VEL
LIN {X 0,Y 459.311,Z 857.28,A -85,B 0,C 180,E1 7755.309,E2 7755.309} C_VEL
LIN {X 0,Y 459.182,Z 857.28,A -85,B 0,C 180,E1 7761.283,E2 7761.283} C_VEL
LIN {X 0,Y 458.989,Z 857.28,A -85,B 0,C 180,E1 7767.519,E2 7767.519} C_VEL
LIN {X 0,Y 458.822,Z 857.28,A -85,B 0,C 180,E1 7774.136,E2 7774.136} C_VEL
LIN {X 0,Y 458.772,Z 857.28,A -85,B 0,C 180,E1 7780.619,E2 7780.619} C_VEL
LIN {X 0,Y 458.879,Z 857.28,A -85,B 0,C 180,E1 7786.552,E2 7786.552} C_VEL
LIN {X 0,Y 458.817,Z 857.28,A -85,B 0,C 180,E1 7792.379,E2 7792.379} C_VEL
LIN {X 0,Y 458.915,Z 857.28,A -85,B 0,C 180,E1 7799.077,E2 7799.077} C_VEL
LIN {X 0,Y 458.915,Z 857.28,A -85,B 0,C 180,E1 7800.253,E2 7800.253} C_VEL
LIN {X 0,Y 459.321,Z 859.926,A -85,B 0,C 180,E1 7800.88,E2 7800.88} C_VEL
LIN {X 0,Y 460.292,Z 869.495,A -85,B 0,C 180,E1 7801.425,E2 7801.425} C_VEL
LIN {X 0,Y 462.41,Z 889.577,A -85,B 0,C 180,E1 7801.87,E2 7801.87} C_VEL
LIN {X 0,Y 465.027,Z 898.12,A -85,B 0,C 180,E1 7802.149,E2 7802.149} C_VEL
LIN {X 0,Y 464.124,Z 939.156,A -85,B 0,C 180,E1 7802.989,E2 7802.989} C_VEL
LIN {X 0,Y 462.048,Z 973.368,A -85,B 0,C 180,E1 7804.413,E2 7804.413} C_VEL
LIN {X 0,Y 459.56,Z 1006.098,A -85,B 0,C 180,E1 7806.584,E2 7806.584} C_VEL
LIN {X 0,Y 457.029,Z 1035.287,A -85,B 0,C 180,E1 7809.391,E2 7809.391} C_VEL
LIN {X 0,Y 454.829,Z 1060.906,A -85,B 0,C 180,E1 7812.817,E2 7812.817} C_VEL
LIN {X 0,Y 453.349,Z 1081.818,A -85,B 0,C 180,E1 7816.727,E2 7816.727} C_VEL
LIN {X 0,Y 452.631,Z 1096.979,A -85,B 0,C 180,E1 7820.918,E2 7820.918} C_VEL
LIN {X 0,Y 452.344,Z 1106.245,A -85,B 0,C 180,E1 7825.201,E2 7825.201} C_VEL
LIN {X 0,Y 452.252,Z 1109.167,A -85,B 0,C 180,E1 7828.082,E2 7828.082} C_VEL
LIN {X 0,Y 452.255,Z 1109.157,A -85,B 0,C 180,E1 7831.919,E2 7831.919} C_VEL
LIN {X 0,Y 452.337,Z 1104.621,A -85,B 0,C 180,E1 7835.764,E2 7835.764} C_VEL
LIN {X 0,Y 452.699,Z 1095.316,A -85,B 0,C 180,E1 7839.627,E2 7839.627} C_VEL
LIN {X 0,Y 453.516,Z 1079.287,A -85,B 0,C 180,E1 7843.791,E2 7843.791} C_VEL
LIN {X 0,Y 455.047,Z 1057.959,A -85,B 0,C 180,E1 7847.612,E2 7847.612} C_VEL
LIN {X 0,Y 457.313,Z 1031.633,A -85,B 0,C 180,E1 7850.977,E2 7850.977} C_VEL
LIN {X 0,Y 459.783,Z 1002.39,A -85,B 0,C 180,E1 7853.663,E2 7853.663} C_VEL
LIN {X 0,Y 462.267,Z 969.763,A -85,B 0,C 180,E1 7855.741,E2 7855.741} C_VEL
LIN {X 0,Y 464.177,Z 935.403,A -85,B 0,C 180,E1 7857.091,E2 7857.091} C_VEL
LIN {X 0,Y 464.253,Z 894.962,A -85,B 0,C 180,E1 7857.915,E2 7857.915} C_VEL
LIN {X 0,Y 451.028,Z 857.28,A -85,B 0,C 180,E1 7859.413,E2 7859.413} C_VEL
LIN {X 0,Y 450.865,Z 857.28,A -85,B 0,C 180,E1 7866.289,E2 7866.289} C_VEL
LIN {X 0,Y 450.769,Z 857.28,A -85,B 0,C 180,E1 7872.348,E2 7872.348} C_VEL
LIN {X 0,Y 450.866,Z 857.28,A -85,B 0,C 180,E1 7877.796,E2 7877.796} C_VEL
LIN {X 0,Y 450.909,Z 857.28,A -85,B 0,C 180,E1 7883.697,E2 7883.697} C_VEL
LIN {X 0,Y 450.966,Z 857.28,A -85,B 0,C 180,E1 7889.747,E2 7889.747} C_VEL
LIN {X 0,Y 451.167,Z 857.28,A -85,B 0,C 180,E1 7896.236,E2 7896.236} C_VEL
LIN {X 0,Y 451.317,Z 857.28,A -85,B 0,C 180,E1 7902.408,E2 7902.408} C_VEL
LIN {X 0,Y 451.38,Z 857.28,A -85,B 0,C 180,E1 7908.369,E2 7908.369} C_VEL
LIN {X 0,Y 451.759,Z 857.28,A -85,B 0,C 180,E1 7914.207,E2 7914.207} C_VEL
LIN {X 0,Y 451.961,Z 857.28,A -85,B 0,C 180,E1 7919.975,E2 7919.975} C_VEL
LIN {X 0,Y 451.711,Z 857.28,A -85,B 0,C 180,E1 7925.744,E2 7925.744} C_VEL
LIN {X 0,Y 451.471,Z 857.28,A -85,B 0,C 180,E1 7931.578,E2 7931.578} C_VEL
LIN {X 0,Y 451.366,Z 857.28,A -85,B 0,C 180,E1 7937.538,E2 7937.538} C_VEL
LIN {X 0,Y 451.137,Z 857.28,A -85,B 0,C 180,E1 7943.712,E2 7943.712} C_VEL
LIN {X 0,Y 450.994,Z 857.28,A -85,B 0,C 180,E1 7950.194,E2 7950.194} C_VEL
LIN {X 0,Y 450.85,Z 857.28,A -85,B 0,C 180,E1 7957.142,E2 7957.142} C_VEL
LIN {X 0,Y 450.806,Z 857.28,A -85,B 0,C 180,E1 7962.362,E2 7962.362} C_VEL
LIN {X 0,Y 450.861,Z 857.28,A -85,B 0,C 180,E1 7967.805,E2 7967.805} C_VEL
LIN {X 0,Y 451.034,Z 857.28,A -85,B 0,C 180,E1 7972.357,E2 7972.357} C_VEL
LIN {X 0,Y 459.083,Z 884.742,A -85,B 0,C 180,E1 7974.296,E2 7974.296} C_VEL
LIN {X 0,Y 460.04,Z 896.448,A -85,B 0,C 180,E1 7975.212,E2 7975.212} C_VEL
LIN {X 0,Y 458.119,Z 920.334,A -85,B 0,C 180,E1 7977.444,E2 7977.444} C_VEL
LIN {X 0,Y 456.238,Z 940.123,A -85,B 0,C 180,E1 7980.145,E2 7980.145} C_VEL
LIN {X 0,Y 454.789,Z 955.36,A -85,B 0,C 180,E1 7983.182,E2 7983.182} C_VEL
LIN {X 0,Y 453.718,Z 967.095,A -85,B 0,C 180,E1 7986.914,E2 7986.914} C_VEL
LIN {X 0,Y 453.12,Z 972.725,A -85,B 0,C 180,E1 7990.479,E2 7990.479} C_VEL
LIN {X 0,Y 452.965,Z 973.235,A -85,B 0,C 180,E1 7994.489,E2 7994.489} C_VEL
LIN {X 0,Y 453.507,Z 967.745,A -85,B 0,C 180,E1 7998.444,E2 7998.444} C_VEL
LIN {X 0,Y 454.329,Z 957.68,A -85,B 0,C 180,E1 8001.857,E2 8001.857} C_VEL
LIN {X 0,Y 455.636,Z 941.737,A -85,B 0,C 180,E1 8005.209,E2 8005.209} C_VEL
LIN {X 0,Y 457.422,Z 921.029,A -85,B 0,C 180,E1 8008.102,E2 8008.102} C_VEL
LIN {X 0,Y 459.281,Z 895.795,A -85,B 0,C 180,E1 8010.472,E2 8010.472} C_VEL
LIN {X 0,Y 458.453,Z 884.862,A -85,B 0,C 180,E1 8011.3,E2 8011.3} C_VEL
LIN {X 0,Y 451.761,Z 857.28,A -85,B 0,C 180,E1 8013.193,E2 8013.193} C_VEL
LIN {X 0,Y 451.592,Z 857.28,A -85,B 0,C 180,E1 8019.65,E2 8019.65} C_VEL
LIN {X 0,Y 451.384,Z 857.28,A -85,B 0,C 180,E1 8025.565,E2 8025.565} C_VEL
LIN {X 0,Y 451.186,Z 857.28,A -85,B 0,C 180,E1 8031.662,E2 8031.662} C_VEL
LIN {X 0,Y 450.974,Z 857.28,A -85,B 0,C 180,E1 8038.035,E2 8038.035} C_VEL
LIN {X 0,Y 450.861,Z 857.28,A -85,B 0,C 180,E1 8044.812,E2 8044.812} C_VEL
LIN {X 0,Y 450.809,Z 857.28,A -85,B 0,C 180,E1 8049.652,E2 8049.652} C_VEL
LIN {X 0,Y 450.816,Z 857.28,A -85,B 0,C 180,E1 8055.206,E2 8055.206} C_VEL
LIN {X 0,Y 451.122,Z 857.28,A -85,B 0,C 180,E1 8058.776,E2 8058.776} C_VEL
LIN {X 0,Y 457.588,Z 886.693,A -85,B 0,C 180,E1 8060.482,E2 8060.482} C_VEL
LIN {X 0,Y 456.805,Z 911.987,A -85,B 0,C 180,E1 8062.462,E2 8062.462} C_VEL
LIN {X 0,Y 455.373,Z 934.577,A -85,B 0,C 180,E1 8065.098,E2 8065.098} C_VEL
LIN {X 0,Y 454.276,Z 951.982,A -85,B 0,C 180,E1 8068.117,E2 8068.117} C_VEL
LIN {X 0,Y 453.575,Z 964.596,A -85,B 0,C 180,E1 8071.533,E2 8071.533} C_VEL
LIN {X 0,Y 453.172,Z 970.885,A -85,B 0,C 180,E1 8074.432,E2 8074.432} C_VEL
LIN {X 0,Y 452.971,Z 973.092,A -85,B 0,C 180,E1 8076.39,E2 8076.39} C_VEL
LIN {X 0,Y 453.007,Z 973.449,A -85,B 0,C 180,E1 8079.362,E2 8079.362} C_VEL
LIN {X 0,Y 453.515,Z 968.862,A -85,B 0,C 180,E1 8083.048,E2 8083.048} C_VEL
LIN {X 0,Y 454.204,Z 958.844,A -85,B 0,C 180,E1 8086.537,E2 8086.537} C_VEL
LIN {X 0,Y 455.265,Z 943.565,A -85,B 0,C 180,E1 8089.756,E2 8089.756} C_VEL
LIN {X 0,Y 456.681,Z 923.049,A -85,B 0,C 180,E1 8092.588,E2 8092.588} C_VEL
LIN {X 0,Y 458.001,Z 898.764,A -85,B 0,C 180,E1 8094.811,E2 8094.811} C_VEL
LIN {X 0,Y 457.574,Z 881.865,A -85,B 0,C 180,E1 8095.931,E2 8095.931} C_VEL
LIN {X 0,Y 451.875,Z 857.28,A -85,B 0,C 180,E1 8097.349,E2 8097.349} C_VEL
LIN {X 0,Y 451.899,Z 857.28,A -85,B 0,C 180,E1 8103.865,E2 8103.865} C_VEL
LIN {X 0,Y 451.597,Z 857.28,A -85,B 0,C 180,E1 8109.671,E2 8109.671} C_VEL
LIN {X 0,Y 451.383,Z 857.28,A -85,B 0,C 180,E1 8115.584,E2 8115.584} C_VEL
LIN {X 0,Y 451.249,Z 857.28,A -85,B 0,C 180,E1 8121.676,E2 8121.676} C_VEL
LIN {X 0,Y 451.006,Z 857.28,A -85,B 0,C 180,E1 8128.049,E2 8128.049} C_VEL
LIN {X 0,Y 450.878,Z 857.28,A -85,B 0,C 180,E1 8134.824,E2 8134.824} C_VEL
LIN {X 0,Y 450.838,Z 857.28,A -85,B 0,C 180,E1 8139.661,E2 8139.661} C_VEL
LIN {X 0,Y 450.863,Z 857.28,A -85,B 0,C 180,E1 8145.154,E2 8145.154} C_VEL
LIN {X 0,Y 450.935,Z 857.28,A -85,B 0,C 180,E1 8150.565,E2 8150.565} C_VEL
LIN {X 0,Y 450.913,Z 857.28,A -85,B 0,C 180,E1 8157.504,E2 8157.504} C_VEL
LIN {X 0,Y 451.071,Z 857.28,A -85,B 0,C 180,E1 8160.683,E2 8160.683} C_VEL
LIN {X 0,Y 462.41,Z 889.577,A -85,B 0,C 180,E1 8161.87,E2 8161.87} C_VEL
LIN {X 0,Y 462.072,Z 898.085,A -85,B 0,C 180,E1 8161.991,E2 8161.991} C_VEL
LIN {X 0,Y 457.647,Z 912.772,A -85,B 0,C 180,E1 8161.995,E2 8161.995} C_VEL
LIN {X 0,Y 456.307,Z 949.123,A -85,B 0,C 180,E1 8162.967,E2 8162.967} C_VEL
LIN {X 0,Y 453.965,Z 981.767,A -85,B 0,C 180,E1 8164.571,E2 8164.571} C_VEL
LIN {X 0,Y 451.398,Z 1012.704,A -85,B 0,C 180,E1 8166.879,E2 8166.879} C_VEL
LIN {X 0,Y 448.697,Z 1041.073,A -85,B 0,C 180,E1 8169.894,E2 8169.894} C_VEL
LIN {X 0,Y 446.65,Z 1065.537,A -85,B 0,C 180,E1 8173.508,E2 8173.508} C_VEL
LIN {X 0,Y 445.319,Z 1084.69,A -85,B 0,C 180,E1 8177.483,E2 8177.483} C_VEL
LIN {X 0,Y 444.721,Z 1097.78,A -85,B 0,C 180,E1 8181.498,E2 8181.498} C_VEL
LIN {X 0,Y 444.513,Z 1105.067,A -85,B 0,C 180,E1 8185.116,E2 8185.116} C_VEL
LIN {X 0,Y 444.428,Z 1107.995,A -85,B 0,C 180,E1 8188.048,E2 8188.048} C_VEL
LIN {X 0,Y 444.432,Z 1107.979,A -85,B 0,C 180,E1 8191.953,E2 8191.953} C_VEL
LIN {X 0,Y 444.519,Z 1103.419,A -85,B 0,C 180,E1 8195.866,E2 8195.866} C_VEL
LIN {X 0,Y 444.831,Z 1094.063,A -85,B 0,C 180,E1 8199.799,E2 8199.799} C_VEL
LIN {X 0,Y 445.68,Z 1078.159,A -85,B 0,C 180,E1 8203.995,E2 8203.995} C_VEL
LIN {X 0,Y 447.203,Z 1057.74,A -85,B 0,C 180,E1 8207.741,E2 8207.741} C_VEL
LIN {X 0,Y 449.514,Z 1032.281,A -85,B 0,C 180,E1 8211.1,E2 8211.1} C_VEL
LIN {X 0,Y 452.179,Z 1002.21,A -85,B 0,C 180,E1 8213.954,E2 8213.954} C_VEL
LIN {X 0,Y 454.824,Z 969.751,A -85,B 0,C 180,E1 8216.076,E2 8216.076} C_VEL
LIN {X 0,Y 456.884,Z 935.218,A -85,B 0,C 180,E1 8217.47,E2 8217.47} C_VEL
LIN {X 0,Y 457.035,Z 896.918,A -85,B 0,C 180,E1 8218.279,E2 8218.279} C_VEL
LIN {X 0,Y 443.088,Z 857.28,A -85,B 0,C 180,E1 8219.869,E2 8219.869} C_VEL
LIN {X 0,Y 442.933,Z 857.28,A -85,B 0,C 180,E1 8225.53,E2 8225.53} C_VEL
LIN {X 0,Y 442.797,Z 857.28,A -85,B 0,C 180,E1 8231.204,E2 8231.204} C_VEL
LIN {X 0,Y 442.863,Z 857.28,A -85,B 0,C 180,E1 8236.85,E2 8236.85} C_VEL
LIN {X 0,Y 442.944,Z 857.28,A -85,B 0,C 180,E1 8242.015,E2 8242.015} C_VEL
LIN {X 0,Y 442.964,Z 857.28,A -85,B 0,C 180,E1 8248.707,E2 8248.707} C_VEL
LIN {X 0,Y 443.153,Z 857.28,A -85,B 0,C 180,E1 8253.615,E2 8253.615} C_VEL
LIN {X 0,Y 443.397,Z 857.28,A -85,B 0,C 180,E1 8260.016,E2 8260.016} C_VEL
LIN {X 0,Y 443.371,Z 857.28,A -85,B 0,C 180,E1 8266.15,E2 8266.15} C_VEL
LIN {X 0,Y 443.732,Z 857.28,A -85,B 0,C 180,E1 8272.134,E2 8272.134} C_VEL
LIN {X 0,Y 444.055,Z 857.28,A -85,B 0,C 180,E1 8278.022,E2 8278.022} C_VEL
LIN {X 0,Y 443.97,Z 857.28,A -85,B 0,C 180,E1 8283.884,E2 8283.884} C_VEL
LIN {X 0,Y 443.667,Z 857.28,A -85,B 0,C 180,E1 8289.795,E2 8289.795} C_VEL
LIN {X 0,Y 443.462,Z 857.28,A -85,B 0,C 180,E1 8295.818,E2 8295.818} C_VEL
LIN {X 0,Y 443.266,Z 857.28,A -85,B 0,C 180,E1 8302.032,E2 8302.032} C_VEL
LIN {X 0,Y 443.08,Z 857.28,A -85,B 0,C 180,E1 8308.539,E2 8308.539} C_VEL
LIN {X 0,Y 442.936,Z 857.28,A -85,B 0,C 180,E1 8315.48,E2 8315.48} C_VEL
LIN {X 0,Y 442.808,Z 857.28,A -85,B 0,C 180,E1 8321.214,E2 8321.214} C_VEL
LIN {X 0,Y 442.881,Z 857.28,A -85,B 0,C 180,E1 8326.862,E2 8326.862} C_VEL
LIN {X 0,Y 443.114,Z 857.942,A -85,B 0,C 180,E1 8331.851,E2 8331.851} C_VEL
LIN {X 0,Y 451.485,Z 885.293,A -85,B 0,C 180,E1 8333.844,E2 8333.844} C_VEL
LIN {X 0,Y 452.848,Z 896.81,A -85,B 0,C 180,E1 8334.787,E2 8334.787} C_VEL
LIN {X 0,Y 450.817,Z 920.608,A -85,B 0,C 180,E1 8337.017,E2 8337.017} C_VEL
LIN {X 0,Y 448.73,Z 941.181,A -85,B 0,C 180,E1 8339.851,E2 8339.851} C_VEL
LIN {X 0,Y 447.085,Z 957.224,A -85,B 0,C 180,E1 8343.146,E2 8343.146} C_VEL
LIN {X 0,Y 445.989,Z 968.165,A -85,B 0,C 180,E1 8346.72,E2 8346.72} C_VEL
LIN {X 0,Y 445.392,Z 973.675,A -85,B 0,C 180,E1 8350.126,E2 8350.126} C_VEL
LIN {X 0,Y 445.148,Z 974.566,A -85,B 0,C 180,E1 8354.21,E2 8354.21} C_VEL
LIN {X 0,Y 445.673,Z 969.491,A -85,B 0,C 180,E1 8358.238,E2 8358.238} C_VEL
LIN {X 0,Y 446.496,Z 959.87,A -85,B 0,C 180,E1 8361.713,E2 8361.713} C_VEL
LIN {X 0,Y 447.882,Z 944.567,A -85,B 0,C 180,E1 8365.126,E2 8365.126} C_VEL
LIN {X 0,Y 449.665,Z 924.7,A -85,B 0,C 180,E1 8368.07,E2 8368.07} C_VEL
LIN {X 0,Y 451.539,Z 901.043,A -85,B 0,C 180,E1 8370.45,E2 8370.45} C_VEL
LIN {X 0,Y 451.352,Z 888.084,A -85,B 0,C 180,E1 8371.464,E2 8371.464} C_VEL
LIN {X 0,Y 444.22,Z 859.516,A -85,B 0,C 180,E1 8373.401,E2 8373.401} C_VEL
LIN {X 0,Y 443.93,Z 857.28,A -85,B 0,C 180,E1 8373.572,E2 8373.572} C_VEL
LIN {X 0,Y 443.681,Z 857.28,A -85,B 0,C 180,E1 8379.824,E2 8379.824} C_VEL
LIN {X 0,Y 443.443,Z 857.28,A -85,B 0,C 180,E1 8385.851,E2 8385.851} C_VEL
LIN {X 0,Y 443.219,Z 857.28,A -85,B 0,C 180,E1 8392.071,E2 8392.071} C_VEL
LIN {X 0,Y 443.047,Z 857.28,A -85,B 0,C 180,E1 8398.583,E2 8398.583} C_VEL
LIN {X 0,Y 442.923,Z 857.28,A -85,B 0,C 180,E1 8405.529,E2 8405.529} C_VEL
LIN {X 0,Y 442.809,Z 857.28,A -85,B 0,C 180,E1 8411.282,E2 8411.282} C_VEL
LIN {X 0,Y 443.132,Z 857.28,A -85,B 0,C 180,E1 8418.425,E2 8418.425} C_VEL
LIN {X 0,Y 449.923,Z 887.252,A -85,B 0,C 180,E1 8420.182,E2 8420.182} C_VEL
LIN {X 0,Y 449.195,Z 913.227,A -85,B 0,C 180,E1 8422.245,E2 8422.245} C_VEL
LIN {X 0,Y 447.686,Z 935.995,A -85,B 0,C 180,E1 8424.952,E2 8424.952} C_VEL
LIN {X 0,Y 446.565,Z 953.005,A -85,B 0,C 180,E1 8427.953,E2 8427.953} C_VEL
LIN {X 0,Y 445.863,Z 964.977,A -85,B 0,C 180,E1 8431.167,E2 8431.167} C_VEL
LIN {X 0,Y 445.275,Z 972.916,A -85,B 0,C 180,E1 8435.017,E2 8435.017} C_VEL
LIN {X 0,Y 445.162,Z 974.942,A -85,B 0,C 180,E1 8438.066,E2 8438.066} C_VEL
LIN {X 0,Y 445.627,Z 971.992,A -85,B 0,C 180,E1 8442.05,E2 8442.05} C_VEL
LIN {X 0,Y 446.284,Z 963.625,A -85,B 0,C 180,E1 8445.664,E2 8445.664} C_VEL
LIN {X 0,Y 447.331,Z 950.131,A -85,B 0,C 180,E1 8448.976,E2 8448.976} C_VEL
LIN {X 0,Y 448.677,Z 930.988,A -85,B 0,C 180,E1 8452.027,E2 8452.027} C_VEL
LIN {X 0,Y 450.08,Z 908.344,A -85,B 0,C 180,E1 8454.426,E2 8454.426} C_VEL
LIN {X 0,Y 450.537,Z 885.679,A -85,B 0,C 180,E1 8456.071,E2 8456.071} C_VEL
LIN {X 0,Y 444.021,Z 857.28,A -85,B 0,C 180,E1 8457.705,E2 8457.705} C_VEL
LIN {X 0,Y 443.98,Z 857.28,A -85,B 0,C 180,E1 8463.934,E2 8463.934} C_VEL
LIN {X 0,Y 443.682,Z 857.28,A -85,B 0,C 180,E1 8469.845,E2 8469.845} C_VEL
LIN {X 0,Y 443.442,Z 857.28,A -85,B 0,C 180,E1 8475.871,E2 8475.871} C_VEL
LIN {X 0,Y 443.284,Z 857.28,A -85,B 0,C 180,E1 8482.085,E2 8482.085} C_VEL
LIN {X 0,Y 443.062,Z 857.28,A -85,B 0,C 180,E1 8488.597,E2 8488.597} C_VEL
LIN {X 0,Y 442.946,Z 857.28,A -85,B 0,C 180,E1 8495.541,E2 8495.541} C_VEL
LIN {X 0,Y 442.822,Z 857.28,A -85,B 0,C 180,E1 8501.219,E2 8501.219} C_VEL
LIN {X 0,Y 442.906,Z 857.28,A -85,B 0,C 180,E1 8506.867,E2 8506.867} C_VEL
LIN {X 0,Y 442.941,Z 857.28,A -85,B 0,C 180,E1 8512.028,E2 8512.028} C_VEL
LIN {X 0,Y 442.988,Z 857.28,A -85,B 0,C 180,E1 8518.708,E2 8518.708} C_VEL
LIN {X 0,Y 443.12,Z 857.28,A -85,B 0,C 180,E1 8520.208,E2 8520.208} C_VEL
LIN {X 0,Y 457.778,Z 900.668,A -85,B 0,C 180,E1 8521.801,E2 8521.801} C_VEL
LIN {X 0,Y 457.647,Z 912.772,A -85,B 0,C 180,E1 8521.995,E2 8521.995} C_VEL
LIN {X 0,Y 453.529,Z 929.784,A -85,B 0,C 180,E1 8522.159,E2 8522.159} C_VEL
LIN {X 0,Y 449.268,Z 944.408,A -85,B 0,C 180,E1 8522.427,E2 8522.427} C_VEL
LIN {X 0,Y 449.103,Z 946.518,A -85,B 0,C 180,E1 8522.502,E2 8522.502} C_VEL
LIN {X 0,Y 446.666,Z 979.819,A -85,B 0,C 180,E1 8524.125,E2 8524.125} C_VEL
LIN {X 0,Y 443.864,Z 1011.375,A -85,B 0,C 180,E1 8526.494,E2 8526.494} C_VEL
LIN {X 0,Y 441.046,Z 1039.639,A -85,B 0,C 180,E1 8529.53,E2 8529.53} C_VEL
LIN {X 0,Y 438.893,Z 1064.217,A -85,B 0,C 180,E1 8533.208,E2 8533.208} C_VEL
LIN {X 0,Y 437.43,Z 1083.423,A -85,B 0,C 180,E1 8537.253,E2 8537.253} C_VEL
LIN {X 0,Y 436.878,Z 1096.604,A -85,B 0,C 180,E1 8541.355,E2 8541.355} C_VEL
LIN {X 0,Y 436.69,Z 1103.889,A -85,B 0,C 180,E1 8545.028,E2 8545.028} C_VEL
LIN {X 0,Y 436.609,Z 1106.823,A -85,B 0,C 180,E1 8548.013,E2 8548.013} C_VEL
LIN {X 0,Y 436.612,Z 1106.799,A -85,B 0,C 180,E1 8551.988,E2 8551.988} C_VEL
LIN {X 0,Y 436.681,Z 1102.212,A -85,B 0,C 180,E1 8555.971,E2 8555.971} C_VEL
LIN {X 0,Y 436.968,Z 1092.81,A -85,B 0,C 180,E1 8559.977,E2 8559.977} C_VEL
LIN {X 0,Y 437.785,Z 1077.919,A -85,B 0,C 180,E1 8564.011,E2 8564.011} C_VEL
LIN {X 0,Y 439.35,Z 1057.872,A -85,B 0,C 180,E1 8567.81,E2 8567.81} C_VEL
LIN {X 0,Y 441.811,Z 1031.845,A -85,B 0,C 180,E1 8571.354,E2 8571.354} C_VEL
LIN {X 0,Y 444.606,Z 1002.088,A -85,B 0,C 180,E1 8574.255,E2 8574.255} C_VEL
LIN {X 0,Y 447.369,Z 970.003,A -85,B 0,C 180,E1 8576.406,E2 8576.406} C_VEL
LIN {X 0,Y 449.593,Z 935.729,A -85,B 0,C 180,E1 8577.845,E2 8577.845} C_VEL
LIN {X 0,Y 449.781,Z 898.68,A -85,B 0,C 180,E1 8578.672,E2 8578.672} C_VEL
LIN {X 0,Y 435.158,Z 857.28,A -85,B 0,C 180,E1 8580.409,E2 8580.409} C_VEL
LIN {X 0,Y 434.905,Z 857.28,A -85,B 0,C 180,E1 8586.792,E2 8586.792} C_VEL
LIN {X 0,Y 434.881,Z 857.28,A -85,B 0,C 180,E1 8593.008,E2 8593.008} C_VEL
LIN {X 0,Y 434.981,Z 857.28,A -85,B 0,C 180,E1 8598.585,E2 8598.585} C_VEL
LIN {X 0,Y 434.973,Z 857.28,A -85,B 0,C 180,E1 8603.706,E2 8603.706} C_VEL
LIN {X 0,Y 435.062,Z 857.28,A -85,B 0,C 180,E1 8608.517,E2 8608.517} C_VEL
LIN {X 0,Y 435.262,Z 857.28,A -85,B 0,C 180,E1 8615.311,E2 8615.311} C_VEL
LIN {X 0,Y 435.465,Z 857.28,A -85,B 0,C 180,E1 8621.746,E2 8621.746} C_VEL
LIN {X 0,Y 435.524,Z 857.28,A -85,B 0,C 180,E1 8627.94,E2 8627.94} C_VEL
LIN {X 0,Y 435.919,Z 857.28,A -85,B 0,C 180,E1 8633.996,E2 8633.996} C_VEL
LIN {X 0,Y 436.165,Z 857.28,A -85,B 0,C 180,E1 8639.975,E2 8639.975} C_VEL
LIN {X 0,Y 435.876,Z 857.28,A -85,B 0,C 180,E1 8645.953,E2 8645.953} C_VEL
LIN {X 0,Y 435.648,Z 857.28,A -85,B 0,C 180,E1 8652.005,E2 8652.005} C_VEL
LIN {X 0,Y 435.473,Z 857.28,A -85,B 0,C 180,E1 8658.2,E2 8658.2} C_VEL
LIN {X 0,Y 435.223,Z 857.28,A -85,B 0,C 180,E1 8665.242,E2 8665.242} C_VEL
LIN {X 0,Y 435.067,Z 857.28,A -85,B 0,C 180,E1 8671.422,E2 8671.422} C_VEL
LIN {X 0,Y 434.895,Z 857.28,A -85,B 0,C 180,E1 8676.798,E2 8676.798} C_VEL
LIN {X 0,Y 434.918,Z 857.28,A -85,B 0,C 180,E1 8683.023,E2 8683.023} C_VEL
LIN {X 0,Y 434.976,Z 857.28,A -85,B 0,C 180,E1 8688.596,E2 8688.596} C_VEL
LIN {X 0,Y 435.091,Z 857.468,A -85,B 0,C 180,E1 8691.258,E2 8691.258} C_VEL
LIN {X 0,Y 443.854,Z 885.556,A -85,B 0,C 180,E1 8693.347,E2 8693.347} C_VEL
LIN {X 0,Y 445.591,Z 898.528,A -85,B 0,C 180,E1 8694.446,E2 8694.446} C_VEL
LIN {X 0,Y 443.281,Z 923.413,A -85,B 0,C 180,E1 8696.872,E2 8696.872} C_VEL
LIN {X 0,Y 441.055,Z 944.024,A -85,B 0,C 180,E1 8699.863,E2 8699.863} C_VEL
LIN {X 0,Y 439.273,Z 960.098,A -85,B 0,C 180,E1 8703.379,E2 8703.379} C_VEL
LIN {X 0,Y 438.195,Z 969.892,A -85,B 0,C 180,E1 8706.818,E2 8706.818} C_VEL
LIN {X 0,Y 437.637,Z 974.55,A -85,B 0,C 180,E1 8709.758,E2 8709.758} C_VEL
LIN {X 0,Y 437.333,Z 975.901,A -85,B 0,C 180,E1 8713.92,E2 8713.92} C_VEL
LIN {X 0,Y 437.839,Z 971.215,A -85,B 0,C 180,E1 8718.024,E2 8718.024} C_VEL
LIN {X 0,Y 438.682,Z 962.028,A -85,B 0,C 180,E1 8721.564,E2 8721.564} C_VEL
LIN {X 0,Y 440.129,Z 947.061,A -85,B 0,C 180,E1 8725.075,E2 8725.075} C_VEL
LIN {X 0,Y 441.911,Z 928.133,A -85,B 0,C 180,E1 8728.036,E2 8728.036} C_VEL
LIN {X 0,Y 444.008,Z 903.925,A -85,B 0,C 180,E1 8730.61,E2 8730.61} C_VEL
LIN {X 0,Y 444.037,Z 890.362,A -85,B 0,C 180,E1 8731.709,E2 8731.709} C_VEL
LIN {X 0,Y 437.153,Z 862.248,A -85,B 0,C 180,E1 8733.691,E2 8733.691} C_VEL
LIN {X 0,Y 436.003,Z 857.28,A -85,B 0,C 180,E1 8733.982,E2 8733.982} C_VEL
LIN {X 0,Y 435.749,Z 857.28,A -85,B 0,C 180,E1 8740.004,E2 8740.004} C_VEL
LIN {X 0,Y 435.531,Z 857.28,A -85,B 0,C 180,E1 8746.147,E2 8746.147} C_VEL
LIN {X 0,Y 435.275,Z 857.28,A -85,B 0,C 180,E1 8752.496,E2 8752.496} C_VEL
LIN {X 0,Y 435.066,Z 857.28,A -85,B 0,C 180,E1 8759.157,E2 8759.157} C_VEL
LIN {X 0,Y 435.01,Z 857.28,A -85,B 0,C 180,E1 8763.84,E2 8763.84} C_VEL
LIN {X 0,Y 434.859,Z 857.28,A -85,B 0,C 180,E1 8770.074,E2 8770.074} C_VEL
LIN {X 0,Y 435.029,Z 857.28,A -85,B 0,C 180,E1 8776.96,E2 8776.96} C_VEL
LIN {X 0,Y 435.216,Z 857.427,A -85,B 0,C 180,E1 8778.104,E2 8778.104} C_VEL
LIN {X 0,Y 441.501,Z 884.638,A -85,B 0,C 180,E1 8779.646,E2 8779.646} C_VEL
LIN {X 0,Y 442.359,Z 900.051,A -85,B 0,C 180,E1 8780.764,E2 8780.764} C_VEL
LIN {X 0,Y 440.826,Z 924.76,A -85,B 0,C 180,E1 8783.133,E2 8783.133} C_VEL
LIN {X 0,Y 439.387,Z 945.771,A -85,B 0,C 180,E1 8786.165,E2 8786.165} C_VEL
LIN {X 0,Y 438.469,Z 960.446,A -85,B 0,C 180,E1 8789.345,E2 8789.345} C_VEL
LIN {X 0,Y 437.864,Z 969.676,A -85,B 0,C 180,E1 8792.468,E2 8792.468} C_VEL
LIN {X 0,Y 437.441,Z 974.692,A -85,B 0,C 180,E1 8795.498,E2 8795.498} C_VEL
LIN {X 0,Y 437.408,Z 975.981,A -85,B 0,C 180,E1 8799.161,E2 8799.161} C_VEL
LIN {X 0,Y 437.934,Z 971.883,A -85,B 0,C 180,E1 8802.944,E2 8802.944} C_VEL
LIN {X 0,Y 438.725,Z 962.41,A -85,B 0,C 180,E1 8806.561,E2 8806.561} C_VEL
LIN {X 0,Y 439.934,Z 947.858,A -85,B 0,C 180,E1 8809.852,E2 8809.852} C_VEL
LIN {X 0,Y 441.441,Z 927.988,A -85,B 0,C 180,E1 8812.812,E2 8812.812} C_VEL
LIN {X 0,Y 442.924,Z 904.724,A -85,B 0,C 180,E1 8815.125,E2 8815.125} C_VEL
LIN {X 0,Y 442.868,Z 886.01,A -85,B 0,C 180,E1 8816.45,E2 8816.45} C_VEL
LIN {X 0,Y 436.16,Z 857.28,A -85,B 0,C 180,E1 8818.161,E2 8818.161} C_VEL
LIN {X 0,Y 436.061,Z 857.28,A -85,B 0,C 180,E1 8824.006,E2 8824.006} C_VEL
LIN {X 0,Y 435.747,Z 857.28,A -85,B 0,C 180,E1 8830.026,E2 8830.026} C_VEL
LIN {X 0,Y 435.544,Z 857.28,A -85,B 0,C 180,E1 8836.166,E2 8836.166} C_VEL
LIN {X 0,Y 435.35,Z 857.28,A -85,B 0,C 180,E1 8842.51,E2 8842.51} C_VEL
LIN {X 0,Y 435.066,Z 857.28,A -85,B 0,C 180,E1 8849.54,E2 8849.54} C_VEL
LIN {X 0,Y 435.057,Z 857.28,A -85,B 0,C 180,E1 8853.851,E2 8853.851} C_VEL
LIN {X 0,Y 434.893,Z 857.28,A -85,B 0,C 180,E1 8860.011,E2 8860.011} C_VEL
LIN {X 0,Y 434.993,Z 857.28,A -85,B 0,C 180,E1 8866.976,E2 8866.976} C_VEL
LIN {X 0,Y 434.965,Z 857.28,A -85,B 0,C 180,E1 8873.719,E2 8873.719} C_VEL
LIN {X 0,Y 435.25,Z 857.958,A -85,B 0,C 180,E1 8879.784,E2 8879.784} C_VEL
LIN {X 0,Y 450.522,Z 901.101,A -85,B 0,C 180,E1 8881.406,E2 8881.406} C_VEL
LIN {X 0,Y 449.435,Z 940.667,A -85,B 0,C 180,E1 8882.29,E2 8882.29} C_VEL
LIN {X 0,Y 449.103,Z 946.518,A -85,B 0,C 180,E1 8882.502,E2 8882.502} C_VEL
LIN {X 0,Y 444.313,Z 962.928,A -85,B 0,C 180,E1 8883.013,E2 8883.013} C_VEL
LIN {X 0,Y 439.551,Z 976.805,A -85,B 0,C 180,E1 8883.602,E2 8883.602} C_VEL
LIN {X 0,Y 439.296,Z 978.764,A -85,B 0,C 180,E1 8883.722,E2 8883.722} C_VEL
LIN {X 0,Y 436.243,Z 1011.155,A -85,B 0,C 180,E1 8886.197,E2 8886.197} C_VEL
LIN {X 0,Y 433.233,Z 1040.175,A -85,B 0,C 180,E1 8889.411,E2 8889.411} C_VEL
LIN {X 0,Y 431.034,Z 1064.296,A -85,B 0,C 180,E1 8893.155,E2 8893.155} C_VEL
LIN {X 0,Y 429.559,Z 1083.172,A -85,B 0,C 180,E1 8897.274,E2 8897.274} C_VEL
LIN {X 0,Y 428.985,Z 1097.052,A -85,B 0,C 180,E1 8901.885,E2 8901.885} C_VEL
LIN {X 0,Y 428.821,Z 1103.998,A -85,B 0,C 180,E1 8905.951,E2 8905.951} C_VEL
LIN {X 0,Y 428.828,Z 1106.259,A -85,B 0,C 180,E1 8910.001,E2 8910.001} C_VEL
LIN {X 0,Y 428.823,Z 1103.936,A -85,B 0,C 180,E1 8914.05,E2 8914.05} C_VEL
LIN {X 0,Y 429.001,Z 1096.927,A -85,B 0,C 180,E1 8918.116,E2 8918.116} C_VEL
LIN {X 0,Y 429.559,Z 1082.936,A -85,B 0,C 180,E1 8922.727,E2 8922.727} C_VEL
LIN {X 0,Y 431.005,Z 1063.93,A -85,B 0,C 180,E1 8926.848,E2 8926.848} C_VEL
LIN {X 0,Y 433.238,Z 1039.719,A -85,B 0,C 180,E1 8930.59,E2 8930.59} C_VEL
LIN {X 0,Y 436.235,Z 1010.718,A -85,B 0,C 180,E1 8933.797,E2 8933.797} C_VEL
LIN {X 0,Y 439.086,Z 979.906,A -85,B 0,C 180,E1 8936.182,E2 8936.182} C_VEL
LIN {X 0,Y 441.718,Z 945.913,A -85,B 0,C 180,E1 8937.902,E2 8937.902} C_VEL
LIN {X 0,Y 443.22,Z 912.619,A -85,B 0,C 180,E1 8938.821,E2 8938.821} C_VEL
LIN {X 0,Y 442.478,Z 900.269,A -85,B 0,C 180,E1 8939.087,E2 8939.087} C_VEL
LIN {X 0,Y 427.185,Z 857.28,A -85,B 0,C 180,E1 8941.016,E2 8941.016} C_VEL
LIN {X 0,Y 426.973,Z 857.28,A -85,B 0,C 180,E1 8947.074,E2 8947.074} C_VEL
LIN {X 0,Y 426.961,Z 857.28,A -85,B 0,C 180,E1 8952.36,E2 8952.36} C_VEL
LIN {X 0,Y 427.043,Z 857.28,A -85,B 0,C 180,E1 8958.122,E2 8958.122} C_VEL
LIN {X 0,Y 427.014,Z 857.28,A -85,B 0,C 180,E1 8964.64,E2 8964.64} C_VEL
LIN {X 0,Y 427.17,Z 857.28,A -85,B 0,C 180,E1 8970.234,E2 8970.234} C_VEL
LIN {X 0,Y 427.409,Z 857.28,A -85,B 0,C 180,E1 8977.08,E2 8977.08} C_VEL
LIN {X 0,Y 427.508,Z 857.28,A -85,B 0,C 180,E1 8983.521,E2 8983.521} C_VEL
LIN {X 0,Y 427.694,Z 857.28,A -85,B 0,C 180,E1 8989.783,E2 8989.783} C_VEL
LIN {X 0,Y 428.01,Z 857.28,A -85,B 0,C 180,E1 8995.919,E2 8995.919} C_VEL
LIN {X 0,Y 428.153,Z 857.28,A -85,B 0,C 180,E1 9002,E2 9002} C_VEL
LIN {X 0,Y 427.888,Z 857.28,A -85,B 0,C 180,E1 9008.107,E2 9008.107} C_VEL
LIN {X 0,Y 427.669,Z 857.28,A -85,B 0,C 180,E1 9014.315,E2 9014.315} C_VEL
LIN {X 0,Y 427.451,Z 857.28,A -85,B 0,C 180,E1 9020.708,E2 9020.708} C_VEL
LIN {X 0,Y 427.206,Z 857.28,A -85,B 0,C 180,E1 9027.619,E2 9027.619} C_VEL
LIN {X 0,Y 427.026,Z 857.28,A -85,B 0,C 180,E1 9034.514,E2 9034.514} C_VEL
LIN {X 0,Y 426.963,Z 857.28,A -85,B 0,C 180,E1 9039.611,E2 9039.611} C_VEL
LIN {X 0,Y 427.041,Z 857.28,A -85,B 0,C 180,E1 9045.1,E2 9045.1} C_VEL
LIN {X 0,Y 427.12,Z 857.614,A -85,B 0,C 180,E1 9050.664,E2 9050.664} C_VEL
LIN {X 0,Y 435.858,Z 884.557,A -85,B 0,C 180,E1 9052.718,E2 9052.718} C_VEL
LIN {X 0,Y 438.425,Z 899.669,A -85,B 0,C 180,E1 9054.049,E2 9054.049} C_VEL
LIN {X 0,Y 435.952,Z 924.616,A -85,B 0,C 180,E1 9056.525,E2 9056.525} C_VEL
LIN {X 0,Y 433.568,Z 945.262,A -85,B 0,C 180,E1 9059.581,E2 9059.581} C_VEL
LIN {X 0,Y 431.595,Z 961.528,A -85,B 0,C 180,E1 9063.222,E2 9063.222} C_VEL
LIN {X 0,Y 430.332,Z 972.22,A -85,B 0,C 180,E1 9067.23,E2 9067.23} C_VEL
LIN {X 0,Y 429.894,Z 975.423,A -85,B 0,C 180,E1 9069.377,E2 9069.377} C_VEL
LIN {X 0,Y 429.523,Z 977.159,A -85,B 0,C 180,E1 9073.62,E2 9073.62} C_VEL
LIN {X 0,Y 429.998,Z 972.934,A -85,B 0,C 180,E1 9077.803,E2 9077.803} C_VEL
LIN {X 0,Y 430.863,Z 964.165,A -85,B 0,C 180,E1 9081.41,E2 9081.41} C_VEL
LIN {X 0,Y 432.262,Z 950.338,A -85,B 0,C 180,E1 9084.869,E2 9084.869} C_VEL
LIN {X 0,Y 434.197,Z 931.503,A -85,B 0,C 180,E1 9088.001,E2 9088.001} C_VEL
LIN {X 0,Y 436.331,Z 908.354,A -85,B 0,C 180,E1 9090.621,E2 9090.621} C_VEL
LIN {X 0,Y 436.652,Z 892.289,A -85,B 0,C 180,E1 9091.986,E2 9091.986} C_VEL
LIN {X 0,Y 429.723,Z 863.539,A -85,B 0,C 180,E1 9094.072,E2 9094.072} C_VEL
LIN {X 0,Y 428.032,Z 857.28,A -85,B 0,C 180,E1 9094.437,E2 9094.437} C_VEL
LIN {X 0,Y 427.826,Z 857.28,A -85,B 0,C 180,E1 9100.191,E2 9100.191} C_VEL
LIN {X 0,Y 427.583,Z 857.28,A -85,B 0,C 180,E1 9106.455,E2 9106.455} C_VEL
LIN {X 0,Y 427.32,Z 857.28,A -85,B 0,C 180,E1 9113.019,E2 9113.019} C_VEL
LIN {X 0,Y 427.14,Z 857.28,A -85,B 0,C 180,E1 9119.752,E2 9119.752} C_VEL
LIN {X 0,Y 426.976,Z 857.28,A -85,B 0,C 180,E1 9127.072,E2 9127.072} C_VEL
LIN {X 0,Y 426.994,Z 857.28,A -85,B 0,C 180,E1 9132.354,E2 9132.354} C_VEL
LIN {X 0,Y 427.266,Z 858.069,A -85,B 0,C 180,E1 9137.762,E2 9137.762} C_VEL
LIN {X 0,Y 433.852,Z 885.563,A -85,B 0,C 180,E1 9139.352,E2 9139.352} C_VEL
LIN {X 0,Y 434.824,Z 900.845,A -85,B 0,C 180,E1 9140.484,E2 9140.484} C_VEL
LIN {X 0,Y 433.193,Z 925.749,A -85,B 0,C 180,E1 9142.9,E2 9142.9} C_VEL
LIN {X 0,Y 431.726,Z 946.433,A -85,B 0,C 180,E1 9145.914,E2 9145.914} C_VEL
LIN {X 0,Y 430.658,Z 962.447,A -85,B 0,C 180,E1 9149.472,E2 9149.472} C_VEL
LIN {X 0,Y 430.014,Z 971.71,A -85,B 0,C 180,E1 9152.801,E2 9152.801} C_VEL
LIN {X 0,Y 429.57,Z 976.683,A -85,B 0,C 180,E1 9156.404,E2 9156.404} C_VEL
LIN {X 0,Y 429.648,Z 977.114,A -85,B 0,C 180,E1 9159.403,E2 9159.403} C_VEL
LIN {X 0,Y 430.128,Z 973.549,A -85,B 0,C 180,E1 9162.798,E2 9162.798} C_VEL
LIN {X 0,Y 430.924,Z 964.994,A -85,B 0,C 180,E1 9166.313,E2 9166.313} C_VEL
LIN {X 0,Y 432.134,Z 951.649,A -85,B 0,C 180,E1 9169.588,E2 9169.588} C_VEL
LIN {X 0,Y 433.606,Z 933.55,A -85,B 0,C 180,E1 9172.532,E2 9172.532} C_VEL
LIN {X 0,Y 435.191,Z 910.567,A -85,B 0,C 180,E1 9175.038,E2 9175.038} C_VEL
LIN {X 0,Y 435.611,Z 888.348,A -85,B 0,C 180,E1 9176.709,E2 9176.709} C_VEL
LIN {X 0,Y 428.756,Z 860.089,A -85,B 0,C 180,E1 9178.382,E2 9178.382} C_VEL
LIN {X 0,Y 428.242,Z 857.28,A -85,B 0,C 180,E1 9178.507,E2 9178.507} C_VEL
LIN {X 0,Y 428.141,Z 857.28,A -85,B 0,C 180,E1 9184.08,E2 9184.08} C_VEL
LIN {X 0,Y 427.812,Z 857.28,A -85,B 0,C 180,E1 9190.214,E2 9190.214} C_VEL
LIN {X 0,Y 427.562,Z 857.28,A -85,B 0,C 180,E1 9197.039,E2 9197.039} C_VEL
LIN {X 0,Y 427.395,Z 857.28,A -85,B 0,C 180,E1 9202.952,E2 9202.952} C_VEL
LIN {X 0,Y 427.172,Z 857.28,A -85,B 0,C 180,E1 9209.766,E2 9209.766} C_VEL
LIN {X 0,Y 426.983,Z 857.28,A -85,B 0,C 180,E1 9217.086,E2 9217.086} C_VEL
LIN {X 0,Y 426.993,Z 857.28,A -85,B 0,C 180,E1 9222.368,E2 9222.368} C_VEL
LIN {X 0,Y 427.069,Z 857.28,A -85,B 0,C 180,E1 9228.128,E2 9228.128} C_VEL
LIN {X 0,Y 427.008,Z 857.28,A -85,B 0,C 180,E1 9234.65,E2 9234.65} C_VEL
LIN {X 0,Y 427.251,Z 857.28,A -85,B 0,C 180,E1 9239.271,E2 9239.271} C_VEL
LIN {X 0,Y 443.271,Z 903.783,A -85,B 0,C 180,E1 9241.047,E2 9241.047} C_VEL
LIN {X 0,Y 442.074,Z 941.354,A -85,B 0,C 180,E1 9241.936,E2 9241.936} C_VEL
LIN {X 0,Y 439.547,Z 975.382,A -85,B 0,C 180,E1 9243.515,E2 9243.515} C_VEL
LIN {X 0,Y 439.296,Z 978.764,A -85,B 0,C 180,E1 9243.722,E2 9243.722} C_VEL
LIN {X 0,Y 434.12,Z 994.335,A -85,B 0,C 180,E1 9244.632,E2 9244.632} C_VEL
LIN {X 0,Y 428.851,Z 1008.694,A -85,B 0,C 180,E1 9245.694,E2 9245.694} C_VEL
LIN {X 0,Y 425.972,Z 1035.785,A -85,B 0,C 180,E1 9248.648,E2 9248.648} C_VEL
LIN {X 0,Y 423.447,Z 1060.085,A -85,B 0,C 180,E1 9252.307,E2 9252.307} C_VEL
LIN {X 0,Y 421.861,Z 1080.085,A -85,B 0,C 180,E1 9256.565,E2 9256.565} C_VEL
LIN {X 0,Y 421.193,Z 1094.155,A -85,B 0,C 180,E1 9261.014,E2 9261.014} C_VEL
LIN {X 0,Y 421.055,Z 1101.535,A -85,B 0,C 180,E1 9264.843,E2 9264.843} C_VEL
LIN {X 0,Y 420.977,Z 1104.48,A -85,B 0,C 180,E1 9267.94,E2 9267.94} C_VEL
LIN {X 0,Y 420.98,Z 1104.442,A -85,B 0,C 180,E1 9272.062,E2 9272.062} C_VEL
LIN {X 0,Y 421.031,Z 1099.801,A -85,B 0,C 180,E1 9276.194,E2 9276.194} C_VEL
LIN {X 0,Y 421.288,Z 1090.304,A -85,B 0,C 180,E1 9280.353,E2 9280.353} C_VEL
LIN {X 0,Y 422.229,Z 1074.116,A -85,B 0,C 180,E1 9284.804,E2 9284.804} C_VEL
LIN {X 0,Y 424.066,Z 1053.522,A -85,B 0,C 180,E1 9288.744,E2 9288.744} C_VEL
LIN {X 0,Y 426.808,Z 1027.185,A -85,B 0,C 180,E1 9292.355,E2 9292.355} C_VEL
LIN {X 0,Y 429.92,Z 997.912,A -85,B 0,C 180,E1 9295.222,E2 9295.222} C_VEL
LIN {X 0,Y 433.06,Z 965.831,A -85,B 0,C 180,E1 9297.386,E2 9297.386} C_VEL
LIN {X 0,Y 435.355,Z 932.311,A -85,B 0,C 180,E1 9298.788,E2 9298.788} C_VEL
LIN {X 0,Y 435.476,Z 902.439,A -85,B 0,C 180,E1 9299.5,E2 9299.5} C_VEL
LIN {X 0,Y 419.279,Z 857.28,A -85,B 0,C 180,E1 9301.56,E2 9301.56} C_VEL
LIN {X 0,Y 419.062,Z 857.28,A -85,B 0,C 180,E1 9307.896,E2 9307.896} C_VEL
LIN {X 0,Y 418.979,Z 857.28,A -85,B 0,C 180,E1 9313.706,E2 9313.706} C_VEL
LIN {X 0,Y 419.081,Z 857.28,A -85,B 0,C 180,E1 9319.421,E2 9319.421} C_VEL
LIN {X 0,Y 419.103,Z 857.28,A -85,B 0,C 180,E1 9326.194,E2 9326.194} C_VEL
LIN {X 0,Y 419.262,Z 857.28,A -85,B 0,C 180,E1 9331.983,E2 9331.983} C_VEL
LIN {X 0,Y 419.542,Z 857.28,A -85,B 0,C 180,E1 9338.826,E2 9338.826} C_VEL
LIN {X 0,Y 419.597,Z 857.28,A -85,B 0,C 180,E1 9345.348,E2 9345.348} C_VEL
LIN {X 0,Y 419.97,Z 857.28,A -85,B 0,C 180,E1 9351.685,E2 9351.685} C_VEL
LIN {X 0,Y 420.346,Z 857.28,A -85,B 0,C 180,E1 9357.91,E2 9357.91} C_VEL
LIN {X 0,Y 420.216,Z 857.28,A -85,B 0,C 180,E1 9364.104,E2 9364.104} C_VEL
LIN {X 0,Y 419.873,Z 857.28,A -85,B 0,C 180,E1 9370.356,E2 9370.356} C_VEL
LIN {X 0,Y 419.708,Z 857.28,A -85,B 0,C 180,E1 9376.739,E2 9376.739} C_VEL
LIN {X 0,Y 419.445,Z 857.28,A -85,B 0,C 180,E1 9383.356,E2 9383.356} C_VEL
LIN {X 0,Y 419.218,Z 857.28,A -85,B 0,C 180,E1 9390.328,E2 9390.328} C_VEL
LIN {X 0,Y 419.066,Z 857.28,A -85,B 0,C 180,E1 9397.357,E2 9397.357} C_VEL
LIN {X 0,Y 419.007,Z 857.28,A -85,B 0,C 180,E1 9403.721,E2 9403.721} C_VEL
LIN {X 0,Y 419.148,Z 857.28,A -85,B 0,C 180,E1 9409.998,E2 9409.998} C_VEL
LIN {X 0,Y 428.851,Z 887.209,A -85,B 0,C 180,E1 9412.379,E2 9412.379} C_VEL
LIN {X 0,Y 431.162,Z 901.918,A -85,B 0,C 180,E1 9413.727,E2 9413.727} C_VEL
LIN {X 0,Y 428.669,Z 925.671,A -85,B 0,C 180,E1 9416.148,E2 9416.148} C_VEL
LIN {X 0,Y 426.135,Z 946.042,A -85,B 0,C 180,E1 9419.201,E2 9419.201} C_VEL
LIN {X 0,Y 424.04,Z 962.146,A -85,B 0,C 180,E1 9422.828,E2 9422.828} C_VEL
LIN {X 0,Y 422.668,Z 972.877,A -85,B 0,C 180,E1 9426.793,E2 9426.793} C_VEL
LIN {X 0,Y 422.203,Z 976.298,A -85,B 0,C 180,E1 9428.984,E2 9428.984} C_VEL
LIN {X 0,Y 421.737,Z 978.396,A -85,B 0,C 180,E1 9433.308,E2 9433.308} C_VEL
LIN {X 0,Y 422.162,Z 974.576,A -85,B 0,C 180,E1 9437.573,E2 9437.573} C_VEL
LIN {X 0,Y 423.065,Z 966.106,A -85,B 0,C 180,E1 9441.279,E2 9441.279} C_VEL
LIN {X 0,Y 424.483,Z 952.373,A -85,B 0,C 180,E1 9444.884,E2 9444.884} C_VEL
LIN {X 0,Y 426.618,Z 932.975,A -85,B 0,C 180,E1 9448.22,E2 9448.22} C_VEL
LIN {X 0,Y 428.845,Z 910.018,A -85,B 0,C 180,E1 9450.884,E2 9450.884} C_VEL
LIN {X 0,Y 429.185,Z 893.831,A -85,B 0,C 180,E1 9452.299,E2 9452.299} C_VEL
LIN {X 0,Y 422.405,Z 865.409,A -85,B 0,C 180,E1 9454.432,E2 9454.432} C_VEL
LIN {X 0,Y 420.095,Z 857.28,A -85,B 0,C 180,E1 9454.91,E2 9454.91} C_VEL
LIN {X 0,Y 419.894,Z 857.28,A -85,B 0,C 180,E1 9460.386,E2 9460.386} C_VEL
LIN {X 0,Y 419.67,Z 857.28,A -85,B 0,C 180,E1 9466.775,E2 9466.775} C_VEL
LIN {X 0,Y 419.386,Z 857.28,A -85,B 0,C 180,E1 9473.398,E2 9473.398} C_VEL
LIN {X 0,Y 419.185,Z 857.28,A -85,B 0,C 180,E1 9480.375,E2 9480.375} C_VEL
LIN {X 0,Y 419.059,Z 857.28,A -85,B 0,C 180,E1 9487.433,E2 9487.433} C_VEL
LIN {X 0,Y 419.014,Z 857.28,A -85,B 0,C 180,E1 9493.788,E2 9493.788} C_VEL
LIN {X 0,Y 419.269,Z 857.28,A -85,B 0,C 180,E1 9497.342,E2 9497.342} C_VEL
LIN {X 0,Y 426.264,Z 887.012,A -85,B 0,C 180,E1 9499.088,E2 9499.088} C_VEL
LIN {X 0,Y 427.308,Z 901.173,A -85,B 0,C 180,E1 9500.157,E2 9500.157} C_VEL
LIN {X 0,Y 425.711,Z 925.035,A -85,B 0,C 180,E1 9502.455,E2 9502.455} C_VEL
LIN {X 0,Y 424.161,Z 945.776,A -85,B 0,C 180,E1 9505.421,E2 9505.421} C_VEL
LIN {X 0,Y 423.008,Z 962.002,A -85,B 0,C 180,E1 9508.911,E2 9508.911} C_VEL
LIN {X 0,Y 422.302,Z 971.849,A -85,B 0,C 180,E1 9512.262,E2 9512.262} C_VEL
